   S702_TL_DC_U262_1.Visu_Adv_Arr[14] := FALSE;
   S702_TL_DC_U262_1.Visu_Adv_Arr[15] := FALSE;
   S702_TL_DC_U262_1.Visu_Ret_Arr[0] := FALSE;
   S702_TL_DC_U262_1.Visu_Ret_Arr[1] := FALSE;
   S702_TL_DC_U262_1.Visu_Ret_Arr[2] := FALSE;
   S702_TL_DC_U262_1.Visu_Ret_Arr[3] := FALSE;
   S702_TL_DC_U262_1.Visu_Ret_Arr[4] := FALSE;
   S702_TL_DC_U262_1.Visu_Ret_Arr[5] := FALSE;
   S702_TL_DC_U262_1.Visu_Ret_Arr[6] := FALSE;
   S702_TL_DC_U262_1.Visu_Ret_Arr[7] := FALSE;
   S702_TL_DC_U262_1.Visu_Ret_Arr[8] := FALSE;
   S702_TL_DC_U262_1.Visu_Ret_Arr[9] := FALSE;
   S702_TL_DC_U262_1.Visu_Ret_Arr[10] := FALSE;
   S702_TL_DC_U262_1.Visu_Ret_Arr[11] := FALSE;
   S702_TL_DC_U262_1.Visu_Ret_Arr[12] := FALSE;
   S702_TL_DC_U262_1.Visu_Ret_Arr[13] := FALSE;
   S702_TL_DC_U262_1.Visu_Ret_Arr[14] := FALSE;
   S702_TL_DC_U262_1.Visu_Ret_Arr[15] := FALSE;
   S702_TL_DC_U262_1.BLK_Move_Ret := 0;
   S702_TL_DC_U262_1.Enable := FALSE;
   S702_TL_DC_U262_1.Adv_End := FALSE;
   S702_TL_DC_U262_1.Ret_End := FALSE;
   S702_TL_DC_U262_1_CLAMP.Enable_Aux := FALSE;
   S702_TL_DC_U262_1_CLAMP.Adv_Amount := 0;
   S702_TL_DC_U262_1_CLAMP.Ret_Amount := 0;
   S702_TL_DC_U262_1_CLAMP.LS_Adv1 := FALSE;
   S702_TL_DC_U262_1_CLAMP.LS_Ret1 := FALSE;
   S702_TL_DC_U262_1_CLAMP.LS_Adv2 := FALSE;
   S702_TL_DC_U262_1_CLAMP.LS_Ret2 := FALSE;
   S702_TL_DC_U262_1_CLAMP.LS_Adv3 := FALSE;
   S702_TL_DC_U262_1_CLAMP.LS_Ret3 := FALSE;
   S702_TL_DC_U262_1_CLAMP.LS_Adv4 := FALSE;
   S702_TL_DC_U262_1_CLAMP.LS_Ret4 := FALSE;
   S702_TL_DC_U262_1_CLAMP.LS_Adv5 := FALSE;
   S702_TL_DC_U262_1_CLAMP.LS_Ret5 := FALSE;
   S702_TL_DC_U262_1_CLAMP.LS_Adv6 := FALSE;
   S702_TL_DC_U262_1_CLAMP.LS_Ret6 := FALSE;
   S702_TL_DC_U262_1_CLAMP.LS_Adv7 := FALSE;
   S702_TL_DC_U262_1_CLAMP.LS_Ret7 := FALSE;
   S702_TL_DC_U262_1_CLAMP.LS_Adv8 := FALSE;
   S702_TL_DC_U262_1_CLAMP.LS_Ret8 := FALSE;
   S702_TL_DC_U262_1_CLAMP.SOL_Adv := FALSE;
   S702_TL_DC_U262_1_CLAMP.SOL_Ret := FALSE;
   S702_TL_DC_U262_1_CLAMP.M_Ready := FALSE;
   S702_TL_DC_U262_1_CLAMP.T_CHK1 := T#0MS;
   S702_TL_DC_U262_1_CLAMP.T_CHK2 := T#0MS;
   S702_TL_DC_U262_1_CLAMP.PB_Lamp_CHK := FALSE;
   S702_TL_DC_U262_1_CLAMP.PB_Error_Rst := FALSE;
   S702_TL_DC_U262_1_CLAMP.M_FLICK := FALSE;
   S702_TL_DC_U262_1_CLAMP.M_Adv_Err := FALSE;
   S702_TL_DC_U262_1_CLAMP.M_Ret_Err := FALSE;
   S702_TL_DC_U262_1_CLAMP.LP_Adv := FALSE;
   S702_TL_DC_U262_1_CLAMP.LP_Ret := FALSE;
   S702_TL_DC_U262_1_CLAMP.Visu_Adv := W#16#0;
   S702_TL_DC_U262_1_CLAMP.Visu_Ret := W#16#0;
   S702_TL_DC_U262_1_CLAMP.Error_T1.IN := FALSE;
   S702_TL_DC_U262_1_CLAMP.Error_T1.PT := T#0MS;
   S702_TL_DC_U262_1_CLAMP.Error_T1.Q := FALSE;
   S702_TL_DC_U262_1_CLAMP.Error_T1.ET := T#0MS;
   S702_TL_DC_U262_1_CLAMP.Error_T1.STATE := B#16#0;
   S702_TL_DC_U262_1_CLAMP.Error_T1.STIME := T#0MS;
   S702_TL_DC_U262_1_CLAMP.Error_T1.ATIME := T#0MS;
   S702_TL_DC_U262_1_CLAMP.Error_T2.IN := FALSE;
   S702_TL_DC_U262_1_CLAMP.Error_T2.PT := T#0MS;
   S702_TL_DC_U262_1_CLAMP.Error_T2.Q := FALSE;
   S702_TL_DC_U262_1_CLAMP.Error_T2.ET := T#0MS;
   S702_TL_DC_U262_1_CLAMP.Error_T2.STATE := B#16#0;
   S702_TL_DC_U262_1_CLAMP.Error_T2.STIME := T#0MS;
   S702_TL_DC_U262_1_CLAMP.Error_T2.ATIME := T#0MS;
   S702_TL_DC_U262_1_CLAMP.Adv_End_Aux := FALSE;
   S702_TL_DC_U262_1_CLAMP.Ret_End_Aux := FALSE;
   S702_TL_DC_U262_1_CLAMP.CHK_Aux1 := FALSE;
   S702_TL_DC_U262_1_CLAMP.CHK_Aux2 := FALSE;
   S702_TL_DC_U262_1_CLAMP.Error_T1_DN := FALSE;
   S702_TL_DC_U262_1_CLAMP.Error_T2_DN := FALSE;
   S702_TL_DC_U262_1_CLAMP.Adv_Memo := FALSE;
   S702_TL_DC_U262_1_CLAMP.Visu_Adv_Arr[0] := FALSE;
   S702_TL_DC_U262_1_CLAMP.Visu_Adv_Arr[1] := FALSE;
   S702_TL_DC_U262_1_CLAMP.Visu_Adv_Arr[2] := FALSE;
   S702_TL_DC_U262_1_CLAMP.Visu_Adv_Arr[3] := FALSE;
   S702_TL_DC_U262_1_CLAMP.Visu_Adv_Arr[4] := FALSE;
   S702_TL_DC_U262_1_CLAMP.Visu_Adv_Arr[5] := FALSE;
   S702_TL_DC_U262_1_CLAMP.Visu_Adv_Arr[6] := FALSE;
   S702_TL_DC_U262_1_CLAMP.Visu_Adv_Arr[7] := FALSE;
   S702_TL_DC_U262_1_CLAMP.Visu_Adv_Arr[8] := FALSE;
   S702_TL_DC_U262_1_CLAMP.Visu_Adv_Arr[9] := FALSE;
   S702_TL_DC_U262_1_CLAMP.Visu_Adv_Arr[10] := FALSE;
   S702_TL_DC_U262_1_CLAMP.Visu_Adv_Arr[11] := FALSE;
   S702_TL_DC_U262_1_CLAMP.Visu_Adv_Arr[12] := FALSE;
   S702_TL_DC_U262_1_CLAMP.Visu_Adv_Arr[13] := FALSE;
   S702_TL_DC_U262_1_CLAMP.Visu_Adv_Arr[14] := FALSE;
   S702_TL_DC_U262_1_CLAMP.Visu_Adv_Arr[15] := FALSE;
   S702_TL_DC_U262_1_CLAMP.Visu_Ret_Arr[0] := FALSE;
   S702_TL_DC_U262_1_CLAMP.Visu_Ret_Arr[1] := FALSE;
   S702_TL_DC_U262_1_CLAMP.Visu_Ret_Arr[2] := FALSE;
   S702_TL_DC_U262_1_CLAMP.Visu_Ret_Arr[3] := FALSE;
   S702_TL_DC_U262_1_CLAMP.Visu_Ret_Arr[4] := FALSE;
   S702_TL_DC_U262_1_CLAMP.Visu_Ret_Arr[5] := FALSE;
   S702_TL_DC_U262_1_CLAMP.Visu_Ret_Arr[6] := FALSE;
   S702_TL_DC_U262_1_CLAMP.Visu_Ret_Arr[7] := FALSE;
   S702_TL_DC_U262_1_CLAMP.Visu_Ret_Arr[8] := FALSE;
   S702_TL_DC_U262_1_CLAMP.Visu_Ret_Arr[9] := FALSE;
   S702_TL_DC_U262_1_CLAMP.Visu_Ret_Arr[10] := FALSE;
   S702_TL_DC_U262_1_CLAMP.Visu_Ret_Arr[11] := FALSE;
   S702_TL_DC_U262_1_CLAMP.Visu_Ret_Arr[12] := FALSE;
   S702_TL_DC_U262_1_CLAMP.Visu_Ret_Arr[13] := FALSE;
   S702_TL_DC_U262_1_CLAMP.Visu_Ret_Arr[14] := FALSE;
   S702_TL_DC_U262_1_CLAMP.Visu_Ret_Arr[15] := FALSE;
   S702_TL_DC_U262_1_CLAMP.BLK_Move_Ret := 0;
   S702_TL_DC_U262_1_CLAMP.Enable := FALSE;
   S702_TL_DC_U262_1_CLAMP.Adv_End := FALSE;
   S702_TL_DC_U262_1_CLAMP.Ret_End := FALSE;
   S702_TL_DC_U261_2_CLAMP.Enable_Aux := FALSE;
   S702_TL_DC_U261_2_CLAMP.Adv_Amount := 0;
   S702_TL_DC_U261_2_CLAMP.Ret_Amount := 0;
   S702_TL_DC_U261_2_CLAMP.LS_Adv1 := FALSE;
   S702_TL_DC_U261_2_CLAMP.LS_Ret1 := FALSE;
   S702_TL_DC_U261_2_CLAMP.LS_Adv2 := FALSE;
   S702_TL_DC_U261_2_CLAMP.LS_Ret2 := FALSE;
   S702_TL_DC_U261_2_CLAMP.LS_Adv3 := FALSE;
   S702_TL_DC_U261_2_CLAMP.LS_Ret3 := FALSE;
   S702_TL_DC_U261_2_CLAMP.LS_Adv4 := FALSE;
   S702_TL_DC_U261_2_CLAMP.LS_Ret4 := FALSE;
   S702_TL_DC_U261_2_CLAMP.LS_Adv5 := FALSE;
   S702_TL_DC_U261_2_CLAMP.LS_Ret5 := FALSE;
   S702_TL_DC_U261_2_CLAMP.LS_Adv6 := FALSE;
   S702_TL_DC_U261_2_CLAMP.LS_Ret6 := FALSE;
   S702_TL_DC_U261_2_CLAMP.LS_Adv7 := FALSE;
   S702_TL_DC_U261_2_CLAMP.LS_Ret7 := FALSE;
   S702_TL_DC_U261_2_CLAMP.LS_Adv8 := FALSE;
   S702_TL_DC_U261_2_CLAMP.LS_Ret8 := FALSE;
   S702_TL_DC_U261_2_CLAMP.SOL_Adv := FALSE;
   S702_TL_DC_U261_2_CLAMP.SOL_Ret := FALSE;
   S702_TL_DC_U261_2_CLAMP.M_Ready := FALSE;
   S702_TL_DC_U261_2_CLAMP.T_CHK1 := T#0MS;
   S702_TL_DC_U261_2_CLAMP.T_CHK2 := T#0MS;
   S702_TL_DC_U261_2_CLAMP.PB_Lamp_CHK := FALSE;
   S702_TL_DC_U261_2_CLAMP.PB_Error_Rst := FALSE;
   S702_TL_DC_U261_2_CLAMP.M_FLICK := FALSE;
   S702_TL_DC_U261_2_CLAMP.M_Adv_Err := FALSE;
   S702_TL_DC_U261_2_CLAMP.M_Ret_Err := FALSE;
   S702_TL_DC_U261_2_CLAMP.LP_Adv := FALSE;
   S702_TL_DC_U261_2_CLAMP.LP_Ret := FALSE;
   S702_TL_DC_U261_2_CLAMP.Visu_Adv := W#16#0;
   S702_TL_DC_U261_2_CLAMP.Visu_Ret := W#16#0;
   S702_TL_DC_U261_2_CLAMP.Error_T1.IN := FALSE;
   S702_TL_DC_U261_2_CLAMP.Error_T1.PT := T#0MS;
   S702_TL_DC_U261_2_CLAMP.Error_T1.Q := FALSE;
   S702_TL_DC_U261_2_CLAMP.Error_T1.ET := T#0MS;
   S702_TL_DC_U261_2_CLAMP.Error_T1.STATE := B#16#0;
   S702_TL_DC_U261_2_CLAMP.Error_T1.STIME := T#0MS;
   S702_TL_DC_U261_2_CLAMP.Error_T1.ATIME := T#0MS;
   S702_TL_DC_U261_2_CLAMP.Error_T2.IN := FALSE;
   S702_TL_DC_U261_2_CLAMP.Error_T2.PT := T#0MS;
   S702_TL_DC_U261_2_CLAMP.Error_T2.Q := FALSE;
   S702_TL_DC_U261_2_CLAMP.Error_T2.ET := T#0MS;
   S702_TL_DC_U261_2_CLAMP.Error_T2.STATE := B#16#0;
   S702_TL_DC_U261_2_CLAMP.Error_T2.STIME := T#0MS;
   S702_TL_DC_U261_2_CLAMP.Error_T2.ATIME := T#0MS;
   S702_TL_DC_U261_2_CLAMP.Adv_End_Aux := FALSE;
   S702_TL_DC_U261_2_CLAMP.Ret_End_Aux := FALSE;
   S702_TL_DC_U261_2_CLAMP.CHK_Aux1 := FALSE;
   S702_TL_DC_U261_2_CLAMP.CHK_Aux2 := FALSE;
   S702_TL_DC_U261_2_CLAMP.Error_T1_DN := FALSE;
   S702_TL_DC_U261_2_CLAMP.Error_T2_DN := FALSE;
   S702_TL_DC_U261_2_CLAMP.Adv_Memo := FALSE;
   S702_TL_DC_U261_2_CLAMP.Visu_Adv_Arr[0] := FALSE;
   S702_TL_DC_U261_2_CLAMP.Visu_Adv_Arr[1] := FALSE;
   S702_TL_DC_U261_2_CLAMP.Visu_Adv_Arr[2] := FALSE;
   S702_TL_DC_U261_2_CLAMP.Visu_Adv_Arr[3] := FALSE;
   S702_TL_DC_U261_2_CLAMP.Visu_Adv_Arr[4] := FALSE;
   S702_TL_DC_U261_2_CLAMP.Visu_Adv_Arr[5] := FALSE;
   S702_TL_DC_U261_2_CLAMP.Visu_Adv_Arr[6] := FALSE;
   S702_TL_DC_U261_2_CLAMP.Visu_Adv_Arr[7] := FALSE;
   S702_TL_DC_U261_2_CLAMP.Visu_Adv_Arr[8] := FALSE;
   S702_TL_DC_U261_2_CLAMP.Visu_Adv_Arr[9] := FALSE;
   S702_TL_DC_U261_2_CLAMP.Visu_Adv_Arr[10] := FALSE;
   S702_TL_DC_U261_2_CLAMP.Visu_Adv_Arr[11] := FALSE;
   S702_TL_DC_U261_2_CLAMP.Visu_Adv_Arr[12] := FALSE;
   S702_TL_DC_U261_2_CLAMP.Visu_Adv_Arr[13] := FALSE;
   S702_TL_DC_U261_2_CLAMP.Visu_Adv_Arr[14] := FALSE;
   S702_TL_DC_U261_2_CLAMP.Visu_Adv_Arr[15] := FALSE;
   S702_TL_DC_U261_2_CLAMP.Visu_Ret_Arr[0] := FALSE;
   S702_TL_DC_U261_2_CLAMP.Visu_Ret_Arr[1] := FALSE;
   S702_TL_DC_U261_2_CLAMP.Visu_Ret_Arr[2] := FALSE;
   S702_TL_DC_U261_2_CLAMP.Visu_Ret_Arr[3] := FALSE;
   S702_TL_DC_U261_2_CLAMP.Visu_Ret_Arr[4] := FALSE;
   S702_TL_DC_U261_2_CLAMP.Visu_Ret_Arr[5] := FALSE;
   S702_TL_DC_U261_2_CLAMP.Visu_Ret_Arr[6] := FALSE;
   S702_TL_DC_U261_2_CLAMP.Visu_Ret_Arr[7] := FALSE;
   S702_TL_DC_U261_2_CLAMP.Visu_Ret_Arr[8] := FALSE;
   S702_TL_DC_U261_2_CLAMP.Visu_Ret_Arr[9] := FALSE;
   S702_TL_DC_U261_2_CLAMP.Visu_Ret_Arr[10] := FALSE;
   S702_TL_DC_U261_2_CLAMP.Visu_Ret_Arr[11] := FALSE;
   S702_TL_DC_U261_2_CLAMP.Visu_Ret_Arr[12] := FALSE;
   S702_TL_DC_U261_2_CLAMP.Visu_Ret_Arr[13] := FALSE;
   S702_TL_DC_U261_2_CLAMP.Visu_Ret_Arr[14] := FALSE;
   S702_TL_DC_U261_2_CLAMP.Visu_Ret_Arr[15] := FALSE;
   S702_TL_DC_U261_2_CLAMP.BLK_Move_Ret := 0;
   S702_TL_DC_U261_2_CLAMP.Enable := FALSE;
   S702_TL_DC_U261_2_CLAMP.Adv_End := FALSE;
   S702_TL_DC_U261_2_CLAMP.Ret_End := FALSE;
END_DATA_BLOCK

FUNCTION FC 124 : VOID
TITLE =
VERSION : 0.1

BEGIN
NETWORK
TITLE =
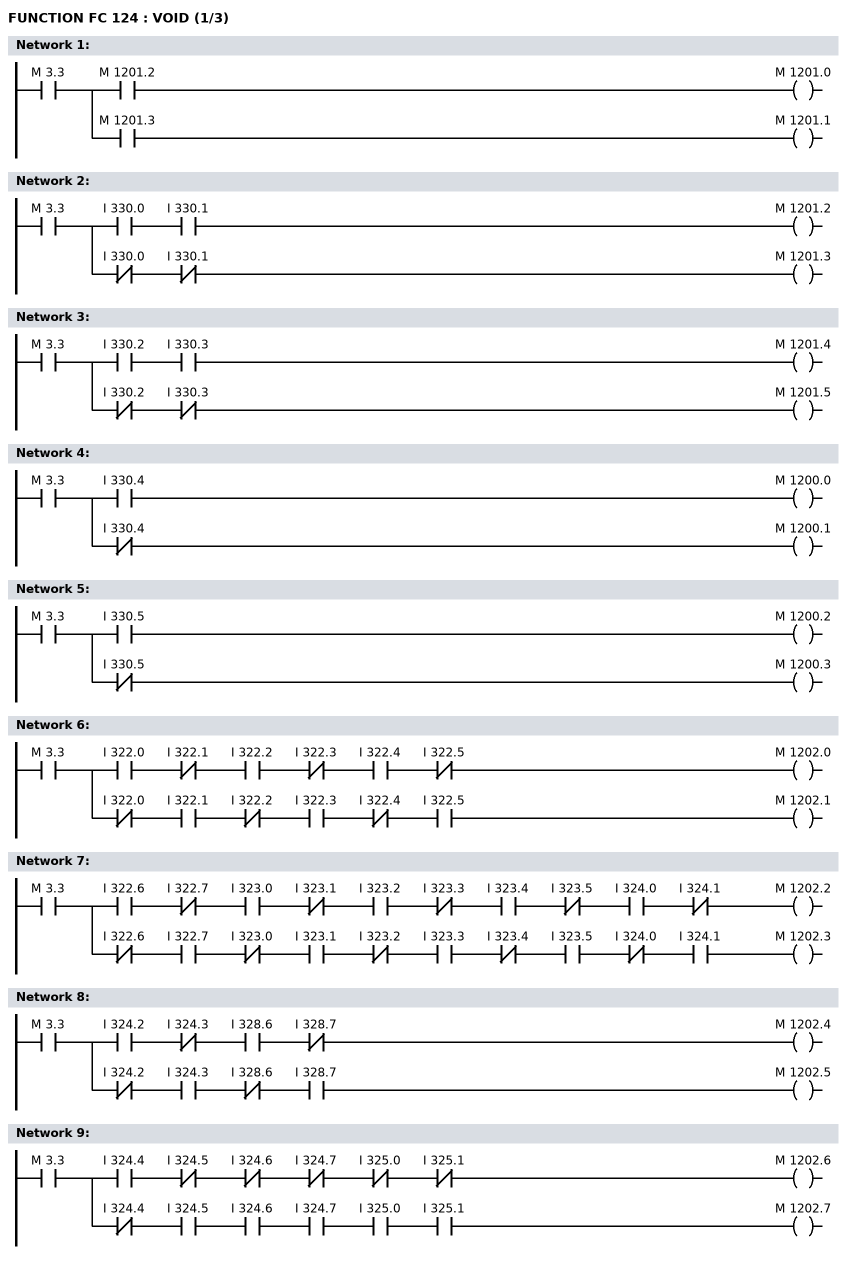

      A     M      3.3;
      =     L      0.0;
      A     L      0.0;
      A     M   1201.2;
      =     M   1201.0;
      A     L      0.0;
      A     M   1201.3;
      =     M   1201.1;
NETWORK
TITLE =

      A     M      3.3;
      =     L      0.0;
      A     L      0.0;
      A     I    330.0;
      A     I    330.1;
      =     M   1201.2;
      A     L      0.0;
      AN    I    330.0;
      AN    I    330.1;
      =     M   1201.3;
NETWORK
TITLE =

      A     M      3.3;
      =     L      0.0;
      A     L      0.0;
      A     I    330.2;
      A     I    330.3;
      =     M   1201.4;
      A     L      0.0;
      AN    I    330.2;
      AN    I    330.3;
      =     M   1201.5;
NETWORK
TITLE =

      A     M      3.3;
      =     L      0.0;
      A     L      0.0;
      A     I    330.4;
      =     M   1200.0;
      A     L      0.0;
      AN    I    330.4;
      =     M   1200.1;
NETWORK
TITLE =

      A     M      3.3;
      =     L      0.0;
      A     L      0.0;
      A     I    330.5;
      =     M   1200.2;
      A     L      0.0;
      AN    I    330.5;
      =     M   1200.3;
NETWORK
TITLE =

      A     M      3.3;
      =     L      0.0;
      A     L      0.0;
      A     I    322.0;
      AN    I    322.1;
      A     I    322.2;
      AN    I    322.3;
      A     I    322.4;
      AN    I    322.5;
      =     M   1202.0;
      A     L      0.0;
      AN    I    322.0;
      A     I    322.1;
      AN    I    322.2;
      A     I    322.3;
      AN    I    322.4;
      A     I    322.5;
      =     M   1202.1;
NETWORK
TITLE =

      A     M      3.3;
      =     L      0.0;
      A     L      0.0;
      A     I    322.6;
      AN    I    322.7;
      A     I    323.0;
      AN    I    323.1;
      A     I    323.2;
      AN    I    323.3;
      A     I    323.4;
      AN    I    323.5;
      A     I    324.0;
      AN    I    324.1;
      =     M   1202.2;
      A     L      0.0;
      AN    I    322.6;
      A     I    322.7;
      AN    I    323.0;
      A     I    323.1;
      AN    I    323.2;
      A     I    323.3;
      AN    I    323.4;
      A     I    323.5;
      AN    I    324.0;
      A     I    324.1;
      =     M   1202.3;
NETWORK
TITLE =

      A     M      3.3;
      =     L      0.0;
      A     L      0.0;
      A     I    324.2;
      AN    I    324.3;
      A     I    328.6;
      AN    I    328.7;
      =     M   1202.4;
      A     L      0.0;
      AN    I    324.2;
      A     I    324.3;
      AN    I    328.6;
      A     I    328.7;
      =     M   1202.5;
NETWORK
TITLE =

      A     M      3.3;
      =     L      0.0;
      A     L      0.0;
      A     I    324.4;
      AN    I    324.5;
      AN    I    324.6;
      AN    I    324.7;
      AN    I    325.0;
      AN    I    325.1;
      =     M   1202.6;
      A     L      0.0;
      AN    I    324.4;
      A     I    324.5;
      A     I    324.6;
      A     I    324.7;
      A     I    325.0;
      A     I    325.1;
      =     M   1202.7;
NETWORK
TITLE =
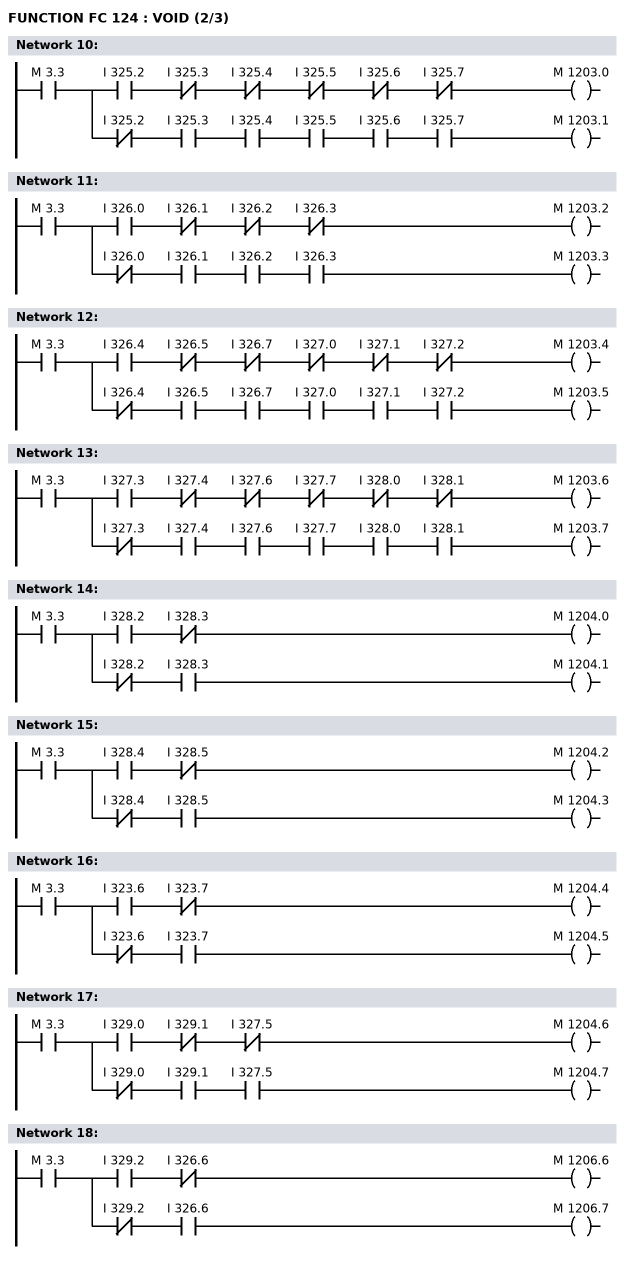

      A     M      3.3;
      =     L      0.0;
      A     L      0.0;
      A     I    325.2;
      AN    I    325.3;
      AN    I    325.4;
      AN    I    325.5;
      AN    I    325.6;
      AN    I    325.7;
      =     M   1203.0;
      A     L      0.0;
      AN    I    325.2;
      A     I    325.3;
      A     I    325.4;
      A     I    325.5;
      A     I    325.6;
      A     I    325.7;
      =     M   1203.1;
NETWORK
TITLE =

      A     M      3.3;
      =     L      0.0;
      A     L      0.0;
      A     I    326.0;
      AN    I    326.1;
      AN    I    326.2;
      AN    I    326.3;
      =     M   1203.2;
      A     L      0.0;
      AN    I    326.0;
      A     I    326.1;
      A     I    326.2;
      A     I    326.3;
      =     M   1203.3;
NETWORK
TITLE =

      A     M      3.3;
      =     L      0.0;
      A     L      0.0;
      A     I    326.4;
      AN    I    326.5;
      AN    I    326.7;
      AN    I    327.0;
      AN    I    327.1;
      AN    I    327.2;
      =     M   1203.4;
      A     L      0.0;
      AN    I    326.4;
      A     I    326.5;
      A     I    326.7;
      A     I    327.0;
      A     I    327.1;
      A     I    327.2;
      =     M   1203.5;
NETWORK
TITLE =

      A     M      3.3;
      =     L      0.0;
      A     L      0.0;
      A     I    327.3;
      AN    I    327.4;
      AN    I    327.6;
      AN    I    327.7;
      AN    I    328.0;
      AN    I    328.1;
      =     M   1203.6;
      A     L      0.0;
      AN    I    327.3;
      A     I    327.4;
      A     I    327.6;
      A     I    327.7;
      A     I    328.0;
      A     I    328.1;
      =     M   1203.7;
NETWORK
TITLE =

      A     M      3.3;
      =     L      0.0;
      A     L      0.0;
      A     I    328.2;
      AN    I    328.3;
      =     M   1204.0;
      A     L      0.0;
      AN    I    328.2;
      A     I    328.3;
      =     M   1204.1;
NETWORK
TITLE =

      A     M      3.3;
      =     L      0.0;
      A     L      0.0;
      A     I    328.4;
      AN    I    328.5;
      =     M   1204.2;
      A     L      0.0;
      AN    I    328.4;
      A     I    328.5;
      =     M   1204.3;
NETWORK
TITLE =

      A     M      3.3;
      =     L      0.0;
      A     L      0.0;
      A     I    323.6;
      AN    I    323.7;
      =     M   1204.4;
      A     L      0.0;
      AN    I    323.6;
      A     I    323.7;
      =     M   1204.5;
NETWORK
TITLE =

      A     M      3.3;
      =     L      0.0;
      A     L      0.0;
      A     I    329.0;
      AN    I    329.1;
      AN    I    327.5;
      =     M   1204.6;
      A     L      0.0;
      AN    I    329.0;
      A     I    329.1;
      A     I    327.5;
      =     M   1204.7;
NETWORK
TITLE =

      A     M      3.3;
      =     L      0.0;
      A     L      0.0;
      A     I    329.2;
      AN    I    326.6;
      =     M   1206.6;
      A     L      0.0;
      AN    I    329.2;
      A     I    326.6;
      =     M   1206.7;
NETWORK
TITLE =
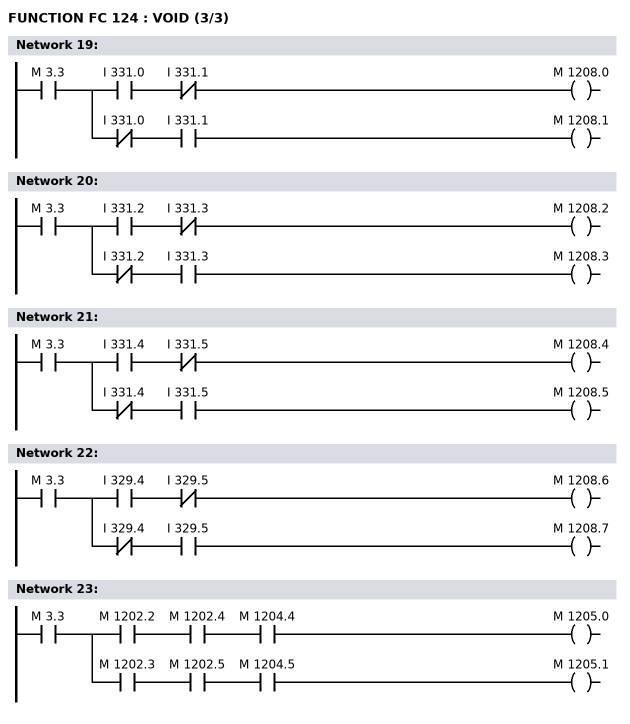

      A     M      3.3;
      =     L      0.0;
      A     L      0.0;
      A     I    331.0;
      AN    I    331.1;
      =     M   1208.0;
      A     L      0.0;
      AN    I    331.0;
      A     I    331.1;
      =     M   1208.1;
NETWORK
TITLE =

      A     M      3.3;
      =     L      0.0;
      A     L      0.0;
      A     I    331.2;
      AN    I    331.3;
      =     M   1208.2;
      A     L      0.0;
      AN    I    331.2;
      A     I    331.3;
      =     M   1208.3;
NETWORK
TITLE =

      A     M      3.3;
      =     L      0.0;
      A     L      0.0;
      A     I    331.4;
      AN    I    331.5;
      =     M   1208.4;
      A     L      0.0;
      AN    I    331.4;
      A     I    331.5;
      =     M   1208.5;
NETWORK
TITLE =

      A     M      3.3;
      =     L      0.0;
      A     L      0.0;
      A     I    329.4;
      AN    I    329.5;
      =     M   1208.6;
      A     L      0.0;
      AN    I    329.4;
      A     I    329.5;
      =     M   1208.7;
NETWORK
TITLE =

      A     M      3.3;
      =     L      0.0;
      A     L      0.0;
      A     M   1202.2;
      A     M   1202.4;
      A     M   1204.4;
      =     M   1205.0;
      A     L      0.0;
      A     M   1202.3;
      A     M   1202.5;
      A     M   1204.5;
      =     M   1205.1;
NETWORK
TITLE =

      A     M      3.3;
      =     L      0.0;
      A     L      0.0;
      A     M   1202.6;
      A     M   1203.0;
      A     M   1203.2;
      A     M   1203.4;
      A     M   1203.6;
      A     M   1206.6;
      =     L      0.1;
      A     L      0.1;
      BLD   102;
      =     M   1205.2;
      A     L      0.1;
      A     M   1204.2;
      A     M   1204.6;
      =     M   1205.4;
      A     L      0.0;
      A     M   1202.7;
      A     M   1203.1;
      A     M   1203.3;
      A     M   1203.5;
      A     M   1203.7;
      A     M   1206.7;
      =     L      0.1;
      A     L      0.1;
      BLD   102;
      =     M   1205.3;
      A     L      0.1;
      A     M   1204.3;
      A     M   1204.7;
      =     M   1205.5;
NETWORK
TITLE =
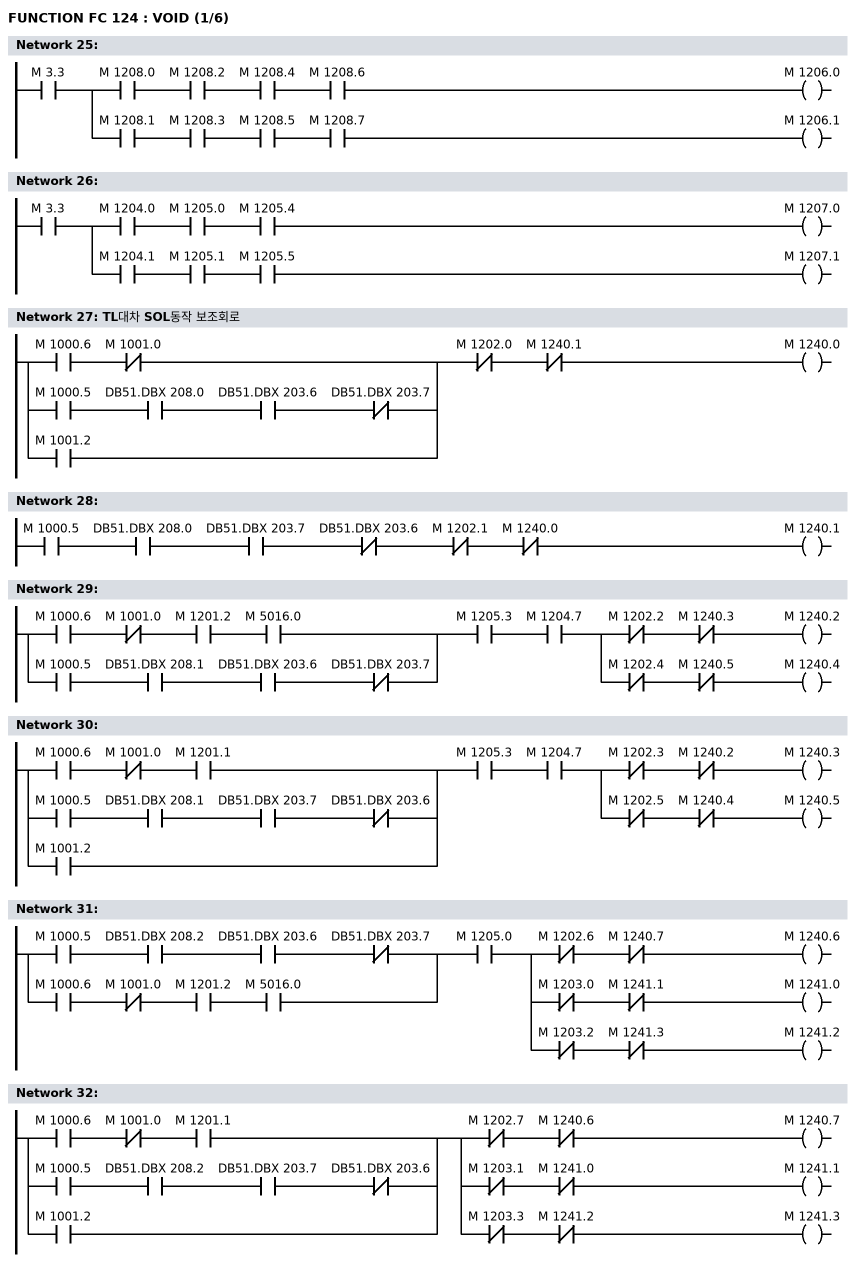

      A     M      3.3;
      =     L      0.0;
      A     L      0.0;
      A     M   1208.0;
      A     M   1208.2;
      A     M   1208.4;
      A     M   1208.6;
      =     M   1206.0;
      A     L      0.0;
      A     M   1208.1;
      A     M   1208.3;
      A     M   1208.5;
      A     M   1208.7;
      =     M   1206.1;
NETWORK
TITLE =

      A     M      3.3;
      =     L      0.0;
      A     L      0.0;
      A     M   1204.0;
      A     M   1205.0;
      A     M   1205.4;
      =     M   1207.0;
      A     L      0.0;
      A     M   1204.1;
      A     M   1205.1;
      A     M   1205.5;
      =     M   1207.1;
NETWORK
TITLE =TL대차 SOL동작 보조회로

      A(    ;
      A     M   1000.6;
      AN    M   1001.0;
      O     ;
      A     M   1000.5;
      A     DB51.DBX  208.0;
      A     DB51.DBX  203.6;
      AN    DB51.DBX  203.7;
      O     M   1001.2;
      )     ;
      AN    M   1202.0;
      AN    M   1240.1;
      =     M   1240.0;
NETWORK
TITLE =

      A     M   1000.5;
      A     DB51.DBX  208.0;
      A     DB51.DBX  203.7;
      AN    DB51.DBX  203.6;
      AN    M   1202.1;
      AN    M   1240.0;
      =     M   1240.1;
NETWORK
TITLE =

      A(    ;
      A     M   1000.6;
      AN    M   1001.0;
      A     M   1201.2;
      A     M   5016.0;
      O     ;
      A     M   1000.5;
      A     DB51.DBX  208.1;
      A     DB51.DBX  203.6;
      AN    DB51.DBX  203.7;
      )     ;
      A     M   1205.3;
      A     M   1204.7;
      =     L      0.0;
      A     L      0.0;
      AN    M   1202.2;
      AN    M   1240.3;
      =     M   1240.2;
      A     L      0.0;
      AN    M   1202.4;
      AN    M   1240.5;
      =     M   1240.4;
NETWORK
TITLE =

      A(    ;
      A     M   1000.6;
      AN    M   1001.0;
      A     M   1201.1;
      O     ;
      A     M   1000.5;
      A     DB51.DBX  208.1;
      A     DB51.DBX  203.7;
      AN    DB51.DBX  203.6;
      O     M   1001.2;
      )     ;
      A     M   1205.3;
      A     M   1204.7;
      =     L      0.0;
      A     L      0.0;
      AN    M   1202.3;
      AN    M   1240.2;
      =     M   1240.3;
      A     L      0.0;
      AN    M   1202.5;
      AN    M   1240.4;
      =     M   1240.5;
NETWORK
TITLE =

      A(    ;
      A     M   1000.5;
      A     DB51.DBX  208.2;
      A     DB51.DBX  203.6;
      AN    DB51.DBX  203.7;
      O     ;
      A     M   1000.6;
      AN    M   1001.0;
      A     M   1201.2;
      A     M   5016.0;
      )     ;
      A     M   1205.0;
      =     L      0.0;
      A     L      0.0;
      AN    M   1202.6;
      AN    M   1240.7;
      =     M   1240.6;
      A     L      0.0;
      AN    M   1203.0;
      AN    M   1241.1;
      =     M   1241.0;
      A     L      0.0;
      AN    M   1203.2;
      AN    M   1241.3;
      =     M   1241.2;
NETWORK
TITLE =

      A     M   1000.6;
      AN    M   1001.0;
      A     M   1201.1;
      O     ;
      A     M   1000.5;
      A     DB51.DBX  208.2;
      A     DB51.DBX  203.7;
      AN    DB51.DBX  203.6;
      O     M   1001.2;
      =     L      0.0;
      A     L      0.0;
      AN    M   1202.7;
      AN    M   1240.6;
      =     M   1240.7;
      A     L      0.0;
      AN    M   1203.1;
      AN    M   1241.0;
      =     M   1241.1;
      A     L      0.0;
      AN    M   1203.3;
      AN    M   1241.2;
      =     M   1241.3;
NETWORK
TITLE =
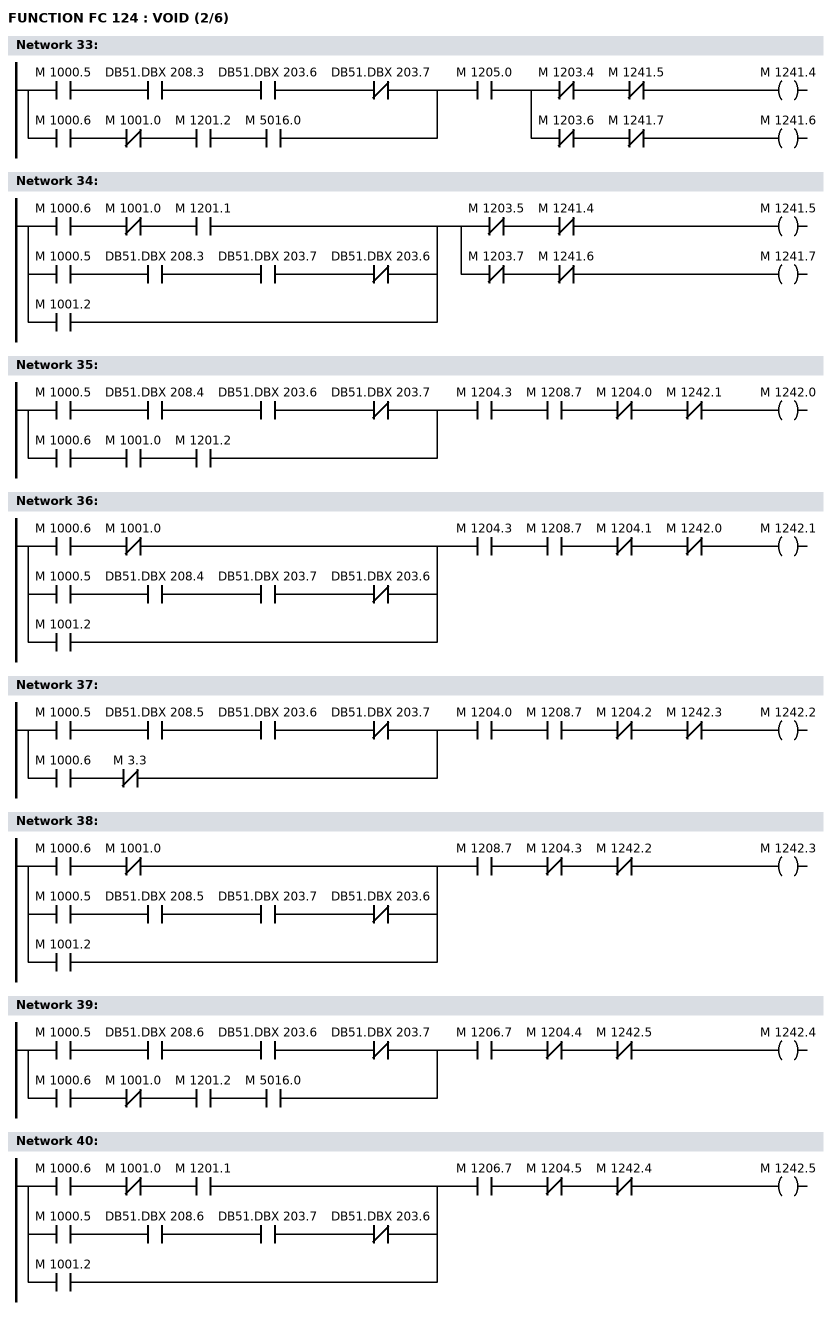

      A(    ;
      A     M   1000.5;
      A     DB51.DBX  208.3;
      A     DB51.DBX  203.6;
      AN    DB51.DBX  203.7;
      O     ;
      A     M   1000.6;
      AN    M   1001.0;
      A     M   1201.2;
      A     M   5016.0;
      )     ;
      A     M   1205.0;
      =     L      0.0;
      A     L      0.0;
      AN    M   1203.4;
      AN    M   1241.5;
      =     M   1241.4;
      A     L      0.0;
      AN    M   1203.6;
      AN    M   1241.7;
      =     M   1241.6;
NETWORK
TITLE =

      A     M   1000.6;
      AN    M   1001.0;
      A     M   1201.1;
      O     ;
      A     M   1000.5;
      A     DB51.DBX  208.3;
      A     DB51.DBX  203.7;
      AN    DB51.DBX  203.6;
      O     M   1001.2;
      =     L      0.0;
      A     L      0.0;
      AN    M   1203.5;
      AN    M   1241.4;
      =     M   1241.5;
      A     L      0.0;
      AN    M   1203.7;
      AN    M   1241.6;
      =     M   1241.7;
NETWORK
TITLE =

      A(    ;
      A     M   1000.5;
      A     DB51.DBX  208.4;
      A     DB51.DBX  203.6;
      AN    DB51.DBX  203.7;
      O     ;
      A     M   1000.6;
      A     M   1001.0;
      A     M   1201.2;
      )     ;
      A     M   1204.3;
      A     M   1208.7;
      AN    M   1204.0;
      AN    M   1242.1;
      =     M   1242.0;
NETWORK
TITLE =

      A(    ;
      A     M   1000.6;
      AN    M   1001.0;
      O     ;
      A     M   1000.5;
      A     DB51.DBX  208.4;
      A     DB51.DBX  203.7;
      AN    DB51.DBX  203.6;
      O     M   1001.2;
      )     ;
      A     M   1204.3;
      A     M   1208.7;
      AN    M   1204.1;
      AN    M   1242.0;
      =     M   1242.1;
NETWORK
TITLE =

      A(    ;
      A     M   1000.5;
      A     DB51.DBX  208.5;
      A     DB51.DBX  203.6;
      AN    DB51.DBX  203.7;
      O     ;
      A     M   1000.6;
      AN    M      3.3;
      )     ;
      A     M   1204.0;
      A     M   1208.7;
      AN    M   1204.2;
      AN    M   1242.3;
      =     M   1242.2;
NETWORK
TITLE =

      A(    ;
      A     M   1000.6;
      AN    M   1001.0;
      O     ;
      A     M   1000.5;
      A     DB51.DBX  208.5;
      A     DB51.DBX  203.7;
      AN    DB51.DBX  203.6;
      O     M   1001.2;
      )     ;
      A     M   1208.7;
      AN    M   1204.3;
      AN    M   1242.2;
      =     M   1242.3;
NETWORK
TITLE =

      A(    ;
      A     M   1000.5;
      A     DB51.DBX  208.6;
      A     DB51.DBX  203.6;
      AN    DB51.DBX  203.7;
      O     ;
      A     M   1000.6;
      AN    M   1001.0;
      A     M   1201.2;
      A     M   5016.0;
      )     ;
      A     M   1206.7;
      AN    M   1204.4;
      AN    M   1242.5;
      =     M   1242.4;
NETWORK
TITLE =

      A(    ;
      A     M   1000.6;
      AN    M   1001.0;
      A     M   1201.1;
      O     ;
      A     M   1000.5;
      A     DB51.DBX  208.6;
      A     DB51.DBX  203.7;
      AN    DB51.DBX  203.6;
      O     M   1001.2;
      )     ;
      A     M   1206.7;
      AN    M   1204.5;
      AN    M   1242.4;
      =     M   1242.5;
NETWORK
TITLE =
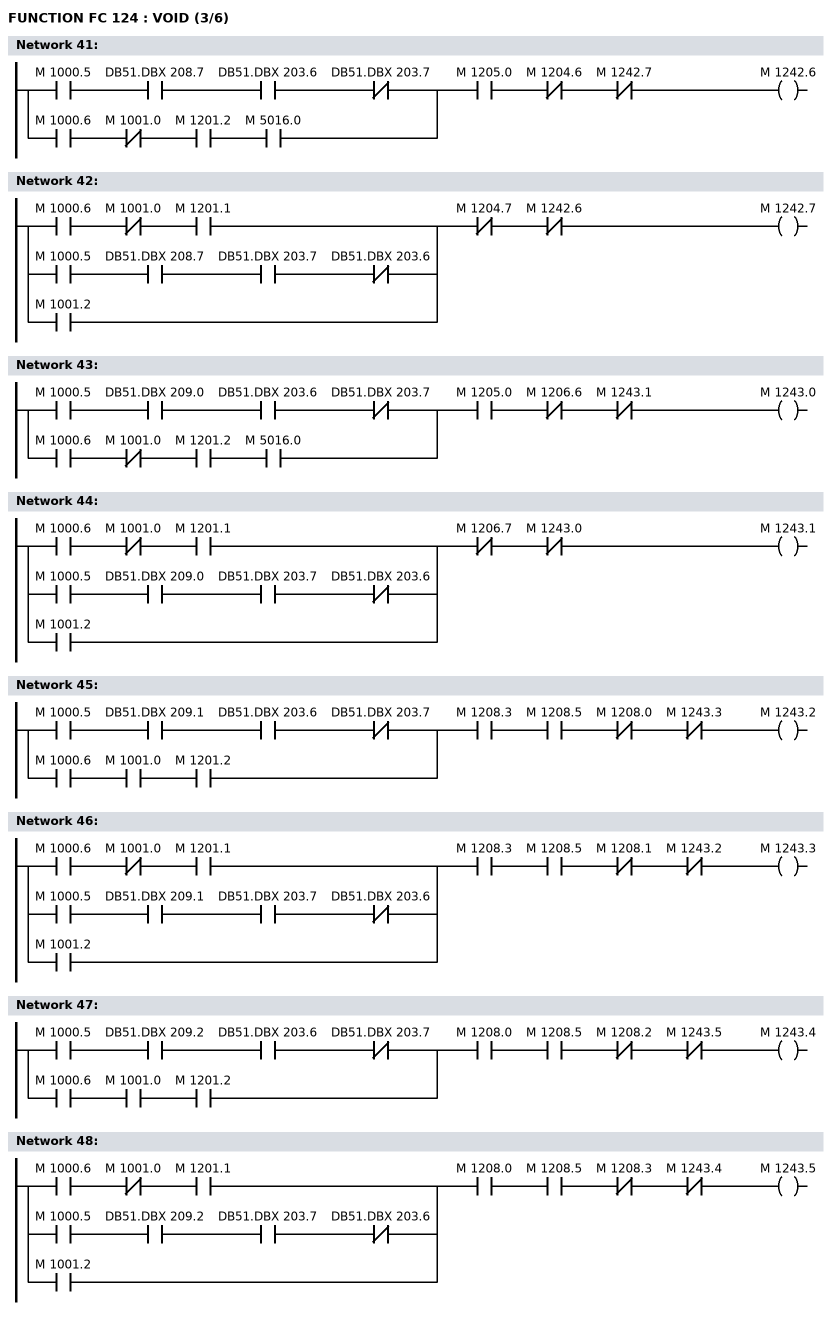

      A(    ;
      A     M   1000.5;
      A     DB51.DBX  208.7;
      A     DB51.DBX  203.6;
      AN    DB51.DBX  203.7;
      O     ;
      A     M   1000.6;
      AN    M   1001.0;
      A     M   1201.2;
      A     M   5016.0;
      )     ;
      A     M   1205.0;
      AN    M   1204.6;
      AN    M   1242.7;
      =     M   1242.6;
NETWORK
TITLE =

      A(    ;
      A     M   1000.6;
      AN    M   1001.0;
      A     M   1201.1;
      O     ;
      A     M   1000.5;
      A     DB51.DBX  208.7;
      A     DB51.DBX  203.7;
      AN    DB51.DBX  203.6;
      O     M   1001.2;
      )     ;
      AN    M   1204.7;
      AN    M   1242.6;
      =     M   1242.7;
NETWORK
TITLE =

      A(    ;
      A     M   1000.5;
      A     DB51.DBX  209.0;
      A     DB51.DBX  203.6;
      AN    DB51.DBX  203.7;
      O     ;
      A     M   1000.6;
      AN    M   1001.0;
      A     M   1201.2;
      A     M   5016.0;
      )     ;
      A     M   1205.0;
      AN    M   1206.6;
      AN    M   1243.1;
      =     M   1243.0;
NETWORK
TITLE =

      A(    ;
      A     M   1000.6;
      AN    M   1001.0;
      A     M   1201.1;
      O     ;
      A     M   1000.5;
      A     DB51.DBX  209.0;
      A     DB51.DBX  203.7;
      AN    DB51.DBX  203.6;
      O     M   1001.2;
      )     ;
      AN    M   1206.7;
      AN    M   1243.0;
      =     M   1243.1;
NETWORK
TITLE =

      A(    ;
      A     M   1000.5;
      A     DB51.DBX  209.1;
      A     DB51.DBX  203.6;
      AN    DB51.DBX  203.7;
      O     ;
      A     M   1000.6;
      A     M   1001.0;
      A     M   1201.2;
      )     ;
      A     M   1208.3;
      A     M   1208.5;
      AN    M   1208.0;
      AN    M   1243.3;
      =     M   1243.2;
NETWORK
TITLE =

      A(    ;
      A     M   1000.6;
      AN    M   1001.0;
      A     M   1201.1;
      O     ;
      A     M   1000.5;
      A     DB51.DBX  209.1;
      A     DB51.DBX  203.7;
      AN    DB51.DBX  203.6;
      O     M   1001.2;
      )     ;
      A     M   1208.3;
      A     M   1208.5;
      AN    M   1208.1;
      AN    M   1243.2;
      =     M   1243.3;
NETWORK
TITLE =

      A(    ;
      A     M   1000.5;
      A     DB51.DBX  209.2;
      A     DB51.DBX  203.6;
      AN    DB51.DBX  203.7;
      O     ;
      A     M   1000.6;
      A     M   1001.0;
      A     M   1201.2;
      )     ;
      A     M   1208.0;
      A     M   1208.5;
      AN    M   1208.2;
      AN    M   1243.5;
      =     M   1243.4;
NETWORK
TITLE =

      A(    ;
      A     M   1000.6;
      AN    M   1001.0;
      A     M   1201.1;
      O     ;
      A     M   1000.5;
      A     DB51.DBX  209.2;
      A     DB51.DBX  203.7;
      AN    DB51.DBX  203.6;
      O     M   1001.2;
      )     ;
      A     M   1208.0;
      A     M   1208.5;
      AN    M   1208.3;
      AN    M   1243.4;
      =     M   1243.5;
NETWORK
TITLE =
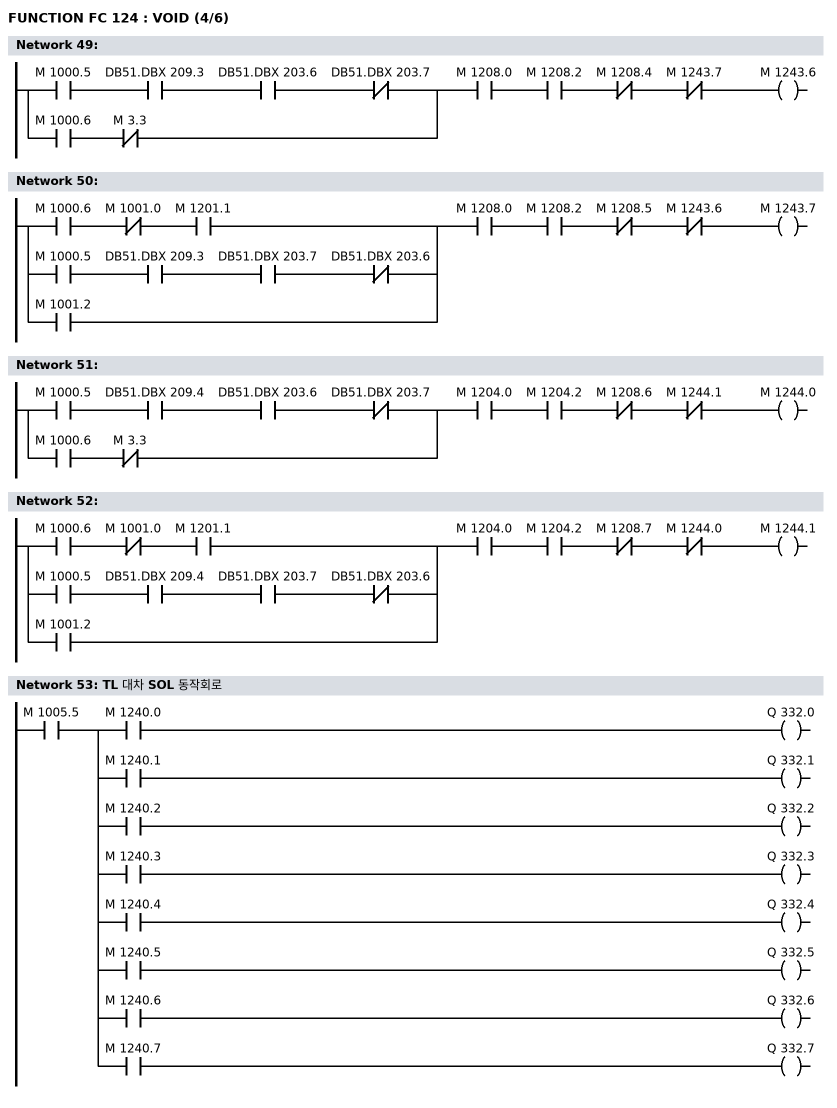

      A(    ;
      A     M   1000.5;
      A     DB51.DBX  209.3;
      A     DB51.DBX  203.6;
      AN    DB51.DBX  203.7;
      O     ;
      A     M   1000.6;
      AN    M      3.3;
      )     ;
      A     M   1208.0;
      A     M   1208.2;
      AN    M   1208.4;
      AN    M   1243.7;
      =     M   1243.6;
NETWORK
TITLE =

      A(    ;
      A     M   1000.6;
      AN    M   1001.0;
      A     M   1201.1;
      O     ;
      A     M   1000.5;
      A     DB51.DBX  209.3;
      A     DB51.DBX  203.7;
      AN    DB51.DBX  203.6;
      O     M   1001.2;
      )     ;
      A     M   1208.0;
      A     M   1208.2;
      AN    M   1208.5;
      AN    M   1243.6;
      =     M   1243.7;
NETWORK
TITLE =

      A(    ;
      A     M   1000.5;
      A     DB51.DBX  209.4;
      A     DB51.DBX  203.6;
      AN    DB51.DBX  203.7;
      O     ;
      A     M   1000.6;
      AN    M      3.3;
      )     ;
      A     M   1204.0;
      A     M   1204.2;
      AN    M   1208.6;
      AN    M   1244.1;
      =     M   1244.0;
NETWORK
TITLE =

      A(    ;
      A     M   1000.6;
      AN    M   1001.0;
      A     M   1201.1;
      O     ;
      A     M   1000.5;
      A     DB51.DBX  209.4;
      A     DB51.DBX  203.7;
      AN    DB51.DBX  203.6;
      O     M   1001.2;
      )     ;
      A     M   1204.0;
      A     M   1204.2;
      AN    M   1208.7;
      AN    M   1244.0;
      =     M   1244.1;
NETWORK
TITLE =TL 대차 SOL 동작회로

      A     M   1005.5;
      =     L      0.0;
      A     L      0.0;
      A     M   1240.0;
      =     Q    332.0;
      A     L      0.0;
      A     M   1240.1;
      =     Q    332.1;
      A     L      0.0;
      A     M   1240.2;
      =     Q    332.2;
      A     L      0.0;
      A     M   1240.3;
      =     Q    332.3;
      A     L      0.0;
      A     M   1240.4;
      =     Q    332.4;
      A     L      0.0;
      A     M   1240.5;
      =     Q    332.5;
      A     L      0.0;
      A     M   1240.6;
      =     Q    332.6;
      A     L      0.0;
      A     M   1240.7;
      =     Q    332.7;
NETWORK
TITLE =
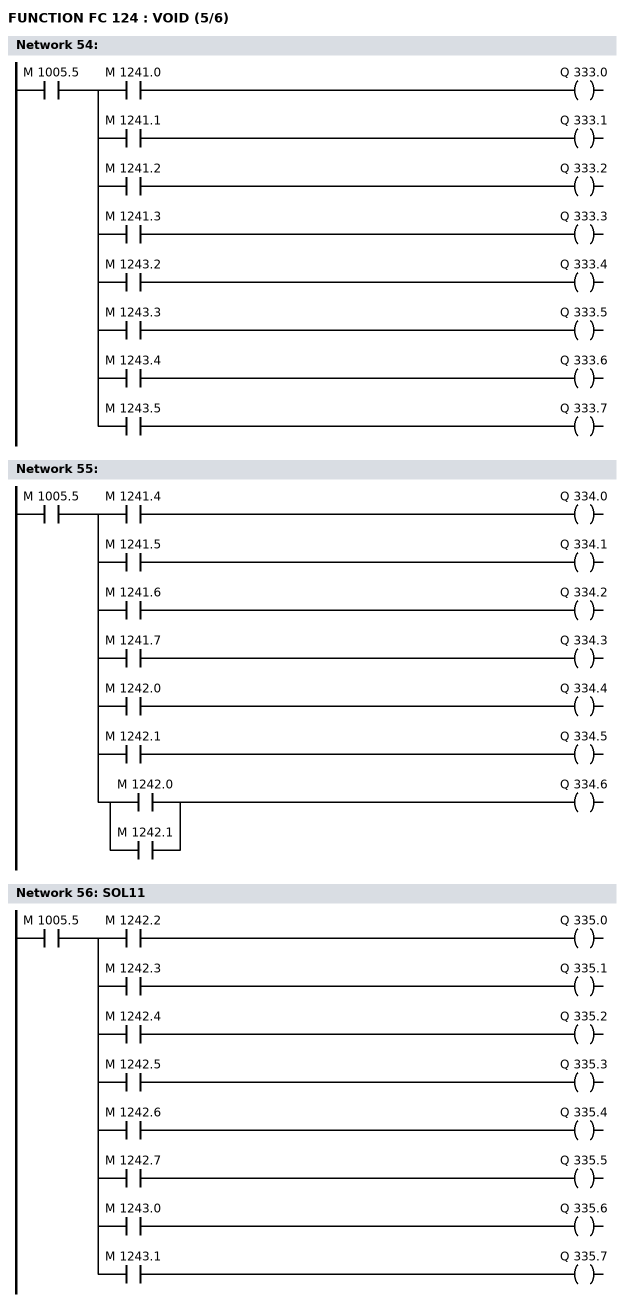

      A     M   1005.5;
      =     L      0.0;
      A     L      0.0;
      A     M   1241.0;
      =     Q    333.0;
      A     L      0.0;
      A     M   1241.1;
      =     Q    333.1;
      A     L      0.0;
      A     M   1241.2;
      =     Q    333.2;
      A     L      0.0;
      A     M   1241.3;
      =     Q    333.3;
      A     L      0.0;
      A     M   1243.2;
      =     Q    333.4;
      A     L      0.0;
      A     M   1243.3;
      =     Q    333.5;
      A     L      0.0;
      A     M   1243.4;
      =     Q    333.6;
      A     L      0.0;
      A     M   1243.5;
      =     Q    333.7;
NETWORK
TITLE =

      A     M   1005.5;
      =     L      0.0;
      A     L      0.0;
      A     M   1241.4;
      =     Q    334.0;
      A     L      0.0;
      A     M   1241.5;
      =     Q    334.1;
      A     L      0.0;
      A     M   1241.6;
      =     Q    334.2;
      A     L      0.0;
      A     M   1241.7;
      =     Q    334.3;
      A     L      0.0;
      A     M   1242.0;
      =     Q    334.4;
      A     L      0.0;
      A     M   1242.1;
      =     Q    334.5;
      A     L      0.0;
      A(    ;
      O     M   1242.0;
      O     M   1242.1;
      )     ;
      =     Q    334.6;
NETWORK
TITLE =SOL11

      A     M   1005.5;
      =     L      0.0;
      A     L      0.0;
      A     M   1242.2;
      =     Q    335.0;
      A     L      0.0;
      A     M   1242.3;
      =     Q    335.1;
      A     L      0.0;
      A     M   1242.4;
      =     Q    335.2;
      A     L      0.0;
      A     M   1242.5;
      =     Q    335.3;
      A     L      0.0;
      A     M   1242.6;
      =     Q    335.4;
      A     L      0.0;
      A     M   1242.7;
      =     Q    335.5;
      A     L      0.0;
      A     M   1243.0;
      =     Q    335.6;
      A     L      0.0;
      A     M   1243.1;
      =     Q    335.7;
NETWORK
TITLE =
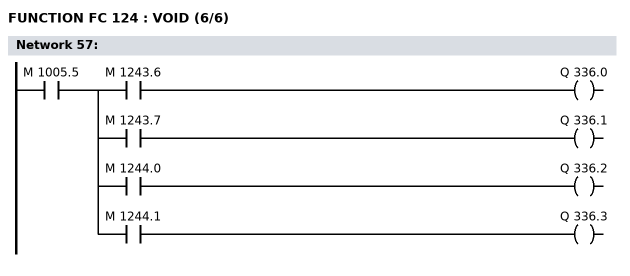

      A     M   1005.5;
      =     L      0.0;
      A     L      0.0;
      A     M   1243.6;
      =     Q    336.0;
      A     L      0.0;
      A     M   1243.7;
      =     Q    336.1;
      A     L      0.0;
      A     M   1244.0;
      =     Q    336.2;
      A     L      0.0;
      A     M   1244.1;
      =     Q    336.3;
END_FUNCTION

FUNCTION FC 125 : VOID
TITLE =
VERSION : 0.1

BEGIN
NETWORK
TITLE =
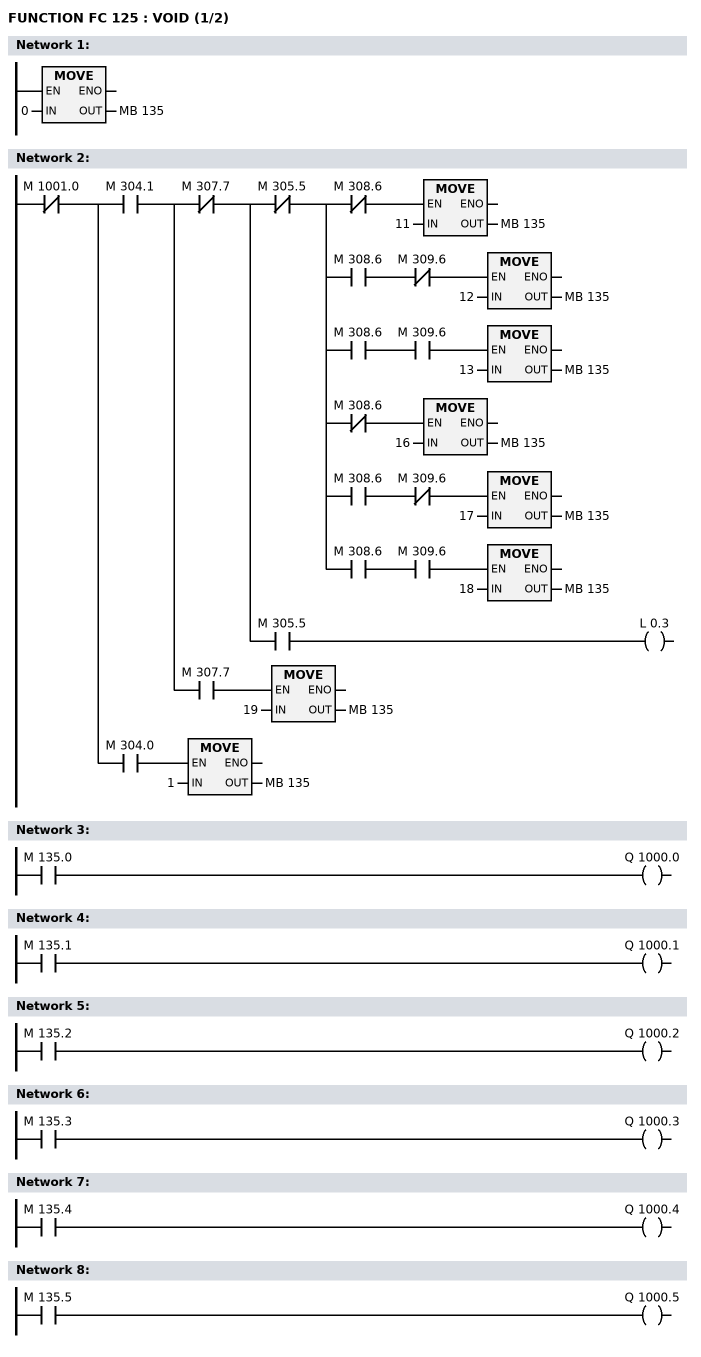

      L     0;
      T     MB   135;
      NOP   0;
NETWORK
TITLE =

      AN    M   1001.0;
      =     L      0.0;
      A     L      0.0;
      A     M    304.1;
      =     L      0.1;
      A     L      0.1;
      AN    M    307.7;
      =     L      0.2;
      A     L      0.2;
      AN    M    305.5;
      =     L      0.3;
      A     L      0.3;
      AN    M    308.6;
      JNB   _001;
      L     11;
      T     MB   135;
_001: NOP   0;
      A     L      0.3;
      A     M    308.6;
      AN    M    309.6;
      JNB   _002;
      L     12;
      T     MB   135;
_002: NOP   0;
      A     L      0.3;
      A     M    308.6;
      A     M    309.6;
      JNB   _003;
      L     13;
      T     MB   135;
_003: NOP   0;
      A     L      0.2;
      A     M    305.5;
      =     L      0.3;
      A     L      0.3;
      AN    M    308.6;
      JNB   _004;
      L     16;
      T     MB   135;
_004: NOP   0;
      A     L      0.3;
      A     M    308.6;
      AN    M    309.6;
      JNB   _005;
      L     17;
      T     MB   135;
_005: NOP   0;
      A     L      0.3;
      A     M    308.6;
      A     M    309.6;
      JNB   _006;
      L     18;
      T     MB   135;
_006: NOP   0;
      A     L      0.1;
      A     M    307.7;
      JNB   _007;
      L     19;
      T     MB   135;
_007: NOP   0;
      A     L      0.0;
      A     M    304.0;
      JNB   _008;
      L     1;
      T     MB   135;
_008: NOP   0;
NETWORK
TITLE =

      A     M    135.0;
      =     Q   1000.0;
NETWORK
TITLE =

      A     M    135.1;
      =     Q   1000.1;
NETWORK
TITLE =

      A     M    135.2;
      =     Q   1000.2;
NETWORK
TITLE =

      A     M    135.3;
      =     Q   1000.3;
NETWORK
TITLE =

      A     M    135.4;
      =     Q   1000.4;
NETWORK
TITLE =

      A     M    135.5;
      =     Q   1000.5;
NETWORK
TITLE =
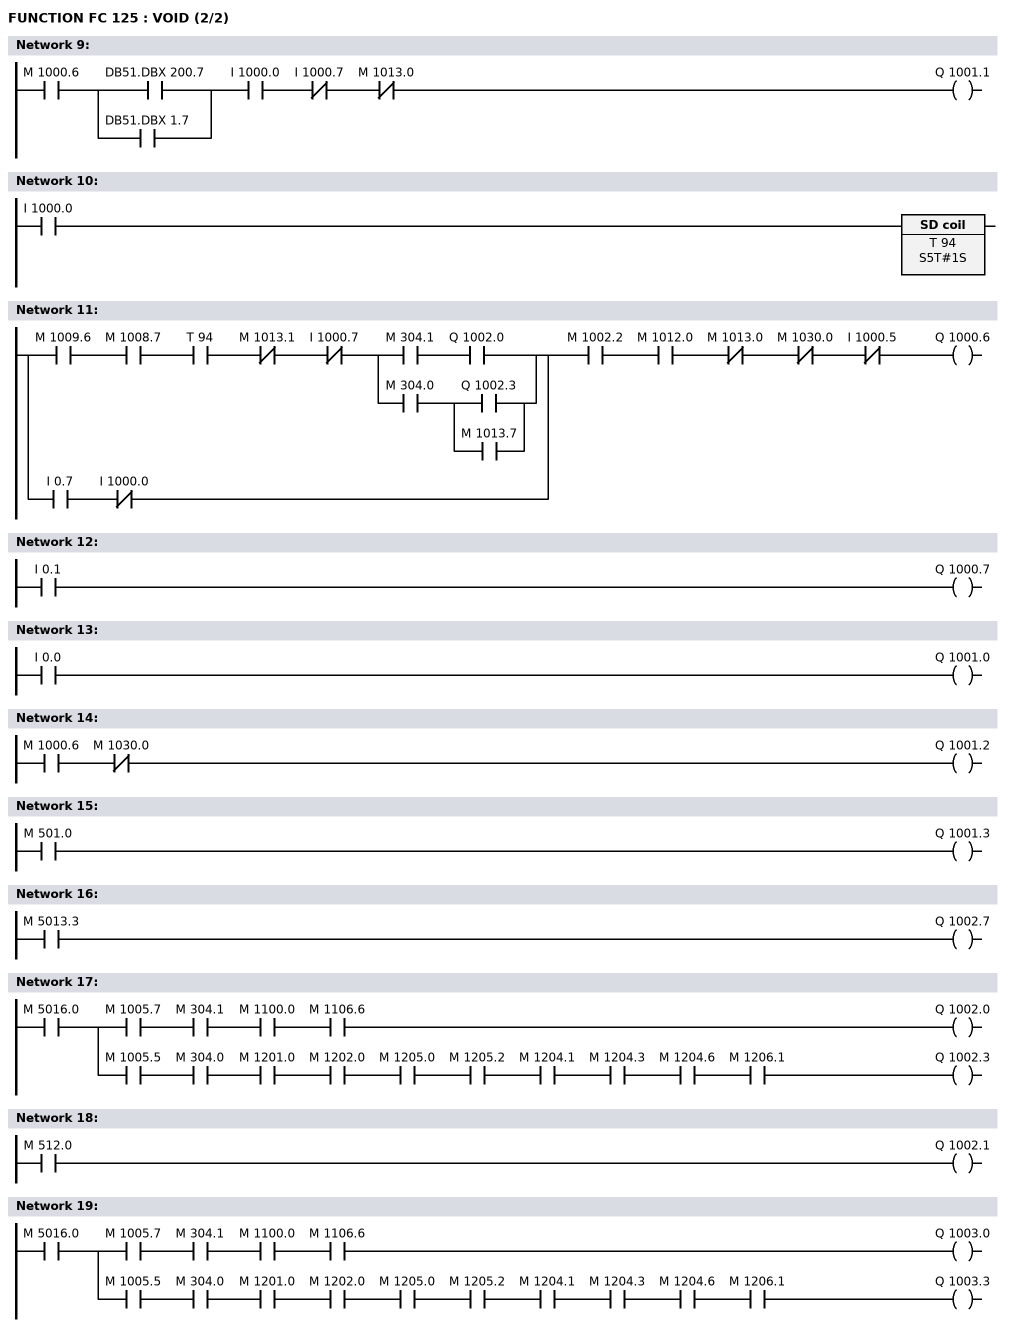

      A     M   1000.6;
      A(    ;
      O     DB51.DBX  200.7;
      O     DB51.DBX    1.7;
      )     ;
      A     I   1000.0;
      AN    I   1000.7;
      AN    M   1013.0;
      =     Q   1001.1;
NETWORK
TITLE =

      A     I   1000.0;
      L     S5T#1S;
      SD    T     94;
NETWORK
TITLE =

      A(    ;
      A     M   1009.6;
      A     M   1008.7;
      A     T     94;
      AN    M   1013.1;
      AN    I   1000.7;
      A(    ;
      A     M    304.1;
      A     Q   1002.0;
      O     ;
      A     M    304.0;
      A(    ;
      O     Q   1002.3;
      O     M   1013.7;
      )     ;
      )     ;
      O     ;
      A     I      0.7;
      AN    I   1000.0;
      )     ;
      A     M   1002.2;
      A     M   1012.0;
      AN    M   1013.0;
      AN    M   1030.0;
      AN    I   1000.5;
      =     Q   1000.6;
NETWORK
TITLE =

      A     I      0.1;
      =     Q   1000.7;
NETWORK
TITLE =

      A     I      0.0;
      =     Q   1001.0;
NETWORK
TITLE =

      A     M   1000.6;
      AN    M   1030.0;
      =     Q   1001.2;
NETWORK
TITLE =

      A     M    501.0;
      =     Q   1001.3;
NETWORK
TITLE =

      A     M   5013.3;
      =     Q   1002.7;
NETWORK
TITLE =

      A     M   5016.0;
      =     L      0.0;
      A     L      0.0;
      A     M   1005.7;
      A     M    304.1;
      A     M   1100.0;
      A     M   1106.6;
      =     Q   1002.0;
      A     L      0.0;
      A     M   1005.5;
      A     M    304.0;
      A     M   1201.0;
      A     M   1202.0;
      A     M   1205.0;
      A     M   1205.2;
      A     M   1204.1;
      A     M   1204.3;
      A     M   1204.6;
      A     M   1206.1;
      =     Q   1002.3;
NETWORK
TITLE =

      A     M    512.0;
      =     Q   1002.1;
NETWORK
TITLE =

      A     M   5016.0;
      =     L      0.0;
      A     L      0.0;
      A     M   1005.7;
      A     M    304.1;
      A     M   1100.0;
      A     M   1106.6;
      =     Q   1003.0;
      A     L      0.0;
      A     M   1005.5;
      A     M    304.0;
      A     M   1201.0;
      A     M   1202.0;
      A     M   1205.0;
      A     M   1205.2;
      A     M   1204.1;
      A     M   1204.3;
      A     M   1204.6;
      A     M   1206.1;
      =     Q   1003.3;
END_FUNCTION

FUNCTION_BLOCK FB 130
TITLE =
VERSION : 0.1


VAR
  S703_MODE : FB 402;
END_VAR
BEGIN
NETWORK
TITLE =
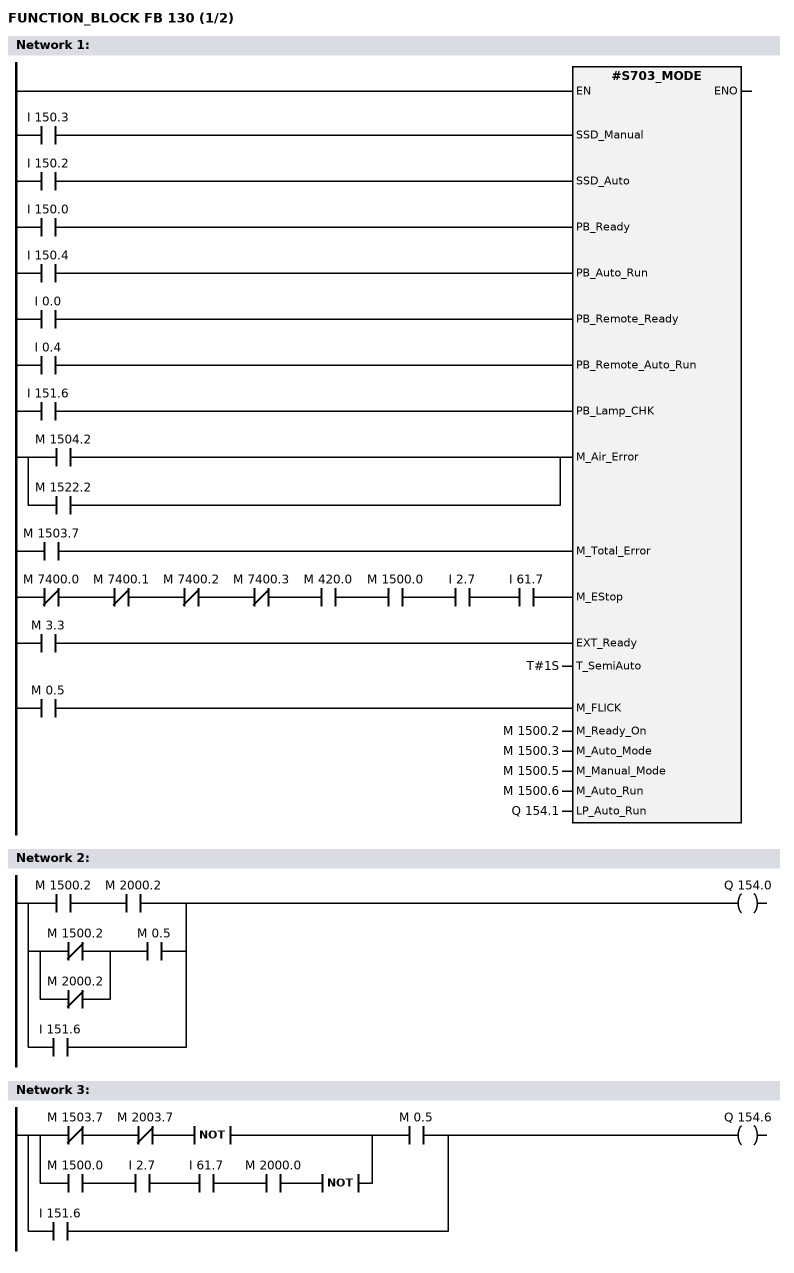

      A     I    150.3;
      =     L      0.0;
      BLD   103;
      A     I    150.2;
      =     L      0.1;
      BLD   103;
      A     I    150.0;
      =     L      0.2;
      BLD   103;
      A     I    150.4;
      =     L      0.3;
      BLD   103;
      A     I      0.0;
      =     L      0.4;
      BLD   103;
      A     I      0.4;
      =     L      0.5;
      BLD   103;
      A     I    151.6;
      =     L      0.6;
      BLD   103;
      A(    ;
      O     M   1504.2;
      O     M   1522.2;
      )     ;
      =     L      0.7;
      BLD   103;
      A     M   1503.7;
      =     L      1.1;
      BLD   103;
      AN    M   7400.0;
      AN    M   7400.1;
      AN    M   7400.2;
      AN    M   7400.3;
      A     M    420.0;
      A     M   1500.0;
      A     I      2.7;
      A     I     61.7;
      =     L      1.2;
      BLD   103;
      A     M      3.3;
      =     L      1.3;
      BLD   103;
      A     M      0.5;
      =     L      1.5;
      BLD   103;
      CALL #S703_MODE (
           SSD_Manual               := L      0.0,
           SSD_Auto                 := L      0.1,
           PB_Ready                 := L      0.2,
           PB_Auto_Run              := L      0.3,
           PB_Remote_Ready          := L      0.4,
           PB_Remote_Auto_Run       := L      0.5,
           PB_Lamp_CHK              := L      0.6,
           M_Air_Error              := L      0.7,
           M_Total_Error            := L      1.1,
           M_EStop                  := L      1.2,
           EXT_Ready                := L      1.3,
           T_SemiAuto               := T#1S,
           M_FLICK                  := L      1.5,
           M_Ready_On               := M   1500.2,
           M_Auto_Mode              := M   1500.3,
           M_Manual_Mode            := M   1500.5,
           M_Auto_Run               := M   1500.6,
           LP_Auto_Run              := Q    154.1);
      NOP   0;
NETWORK
TITLE =

      A     M   1500.2;
      A     M   2000.2;
      O     ;
      A(    ;
      ON    M   1500.2;
      ON    M   2000.2;
      )     ;
      A     M      0.5;
      O     I    151.6;
      =     Q    154.0;
NETWORK
TITLE =

      A(    ;
      AN    M   1503.7;
      AN    M   2003.7;
      NOT   ;
      O(    ;
      A     M   1500.0;
      A     I      2.7;
      A     I     61.7;
      A     M   2000.0;
      NOT   ;
      )     ;
      )     ;
      A     M      0.5;
      O     I    151.6;
      =     Q    154.6;
NETWORK
TITLE =
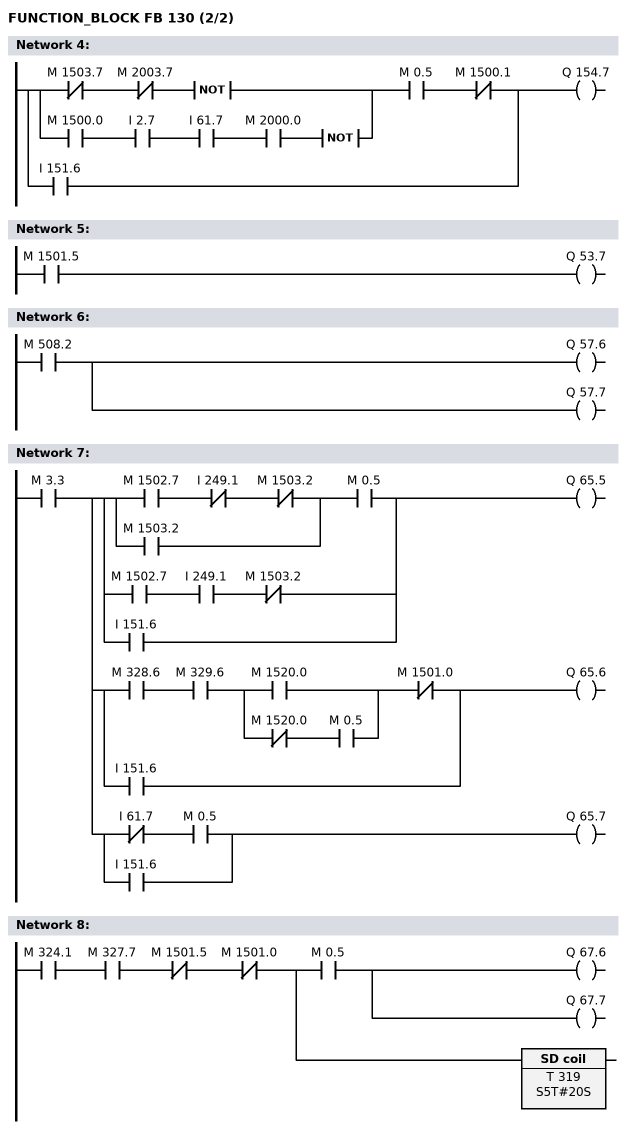

      A(    ;
      AN    M   1503.7;
      AN    M   2003.7;
      NOT   ;
      O(    ;
      A     M   1500.0;
      A     I      2.7;
      A     I     61.7;
      A     M   2000.0;
      NOT   ;
      )     ;
      )     ;
      A     M      0.5;
      AN    M   1500.1;
      O     I    151.6;
      =     Q    154.7;
NETWORK
TITLE =

      A     M   1501.5;
      =     Q     53.7;
NETWORK
TITLE =

      A     M    508.2;
      =     Q     57.6;
      =     Q     57.7;
NETWORK
TITLE =

      A     M      3.3;
      =     L      0.0;
      A     L      0.0;
      A(    ;
      A(    ;
      A     M   1502.7;
      AN    I    249.1;
      AN    M   1503.2;
      O     M   1503.2;
      )     ;
      A     M      0.5;
      O     ;
      A     M   1502.7;
      A     I    249.1;
      AN    M   1503.2;
      O     I    151.6;
      )     ;
      =     Q     65.5;
      A     L      0.0;
      A(    ;
      A     M    328.6;
      A     M    329.6;
      A(    ;
      O     M   1520.0;
      O     ;
      AN    M   1520.0;
      A     M      0.5;
      )     ;
      AN    M   1501.0;
      O     I    151.6;
      )     ;
      =     Q     65.6;
      A     L      0.0;
      A(    ;
      AN    I     61.7;
      A     M      0.5;
      O     I    151.6;
      )     ;
      =     Q     65.7;
NETWORK
TITLE =

      A     M    324.1;
      A     M    327.7;
      AN    M   1501.5;
      AN    M   1501.0;
      =     L      0.0;
      A     L      0.0;
      A     M      0.5;
      =     Q     67.6;
      =     Q     67.7;
      A     L      0.0;
      BLD   102;
      L     S5T#20S;
      SD    T    319;
END_FUNCTION_BLOCK

DATA_BLOCK DB 130
TITLE =
VERSION : 0.0

 FB 130
BEGIN
   S703_MODE.SSD_Manual := FALSE;
   S703_MODE.SSD_Auto := FALSE;
   S703_MODE.PB_Ready := FALSE;
   S703_MODE.PB_Auto_Run := FALSE;
   S703_MODE.PB_Remote_Ready := FALSE;
   S703_MODE.PB_Remote_Auto_Run := FALSE;
   S703_MODE.PB_Lamp_CHK := FALSE;
   S703_MODE.M_Air_Error := FALSE;
   S703_MODE.M_Water_Error := FALSE;
   S703_MODE.M_Total_Error := FALSE;
   S703_MODE.M_EStop := FALSE;
   S703_MODE.EXT_Ready := FALSE;
   S703_MODE.EXT_Auto := FALSE;
   S703_MODE.T_SemiAuto := T#0MS;
   S703_MODE.M_FLICK := FALSE;
   S703_MODE.M_Ready_On := FALSE;
   S703_MODE.M_Auto_Mode := FALSE;
   S703_MODE.M_SemiAuto_Mode := FALSE;
   S703_MODE.M_Manual_Mode := FALSE;
   S703_MODE.M_Auto_Run := FALSE;
   S703_MODE.LP_Ready_On := FALSE;
   S703_MODE.LP_Auto_Run := FALSE;
   S703_MODE.AUTO_MODE_DELAY.IN := FALSE;
   S703_MODE.AUTO_MODE_DELAY.PT := T#0MS;
   S703_MODE.AUTO_MODE_DELAY.Q := FALSE;
   S703_MODE.AUTO_MODE_DELAY.ET := T#0MS;
   S703_MODE.AUTO_MODE_DELAY.STATE := B#16#0;
   S703_MODE.AUTO_MODE_DELAY.STIME := T#0MS;
   S703_MODE.AUTO_MODE_DELAY.ATIME := T#0MS;
   S703_MODE.SEMI_AUTO_DELAY.IN := FALSE;
   S703_MODE.SEMI_AUTO_DELAY.PT := T#0MS;
   S703_MODE.SEMI_AUTO_DELAY.Q := FALSE;
   S703_MODE.SEMI_AUTO_DELAY.ET := T#0MS;
   S703_MODE.SEMI_AUTO_DELAY.STATE := B#16#0;
   S703_MODE.SEMI_AUTO_DELAY.STIME := T#0MS;
   S703_MODE.SEMI_AUTO_DELAY.ATIME := T#0MS;
   S703_MODE.MANUAL_DELAY.IN := FALSE;
   S703_MODE.MANUAL_DELAY.PT := T#0MS;
   S703_MODE.MANUAL_DELAY.Q := FALSE;
   S703_MODE.MANUAL_DELAY.ET := T#0MS;
   S703_MODE.MANUAL_DELAY.STATE := B#16#0;
   S703_MODE.MANUAL_DELAY.STIME := T#0MS;
   S703_MODE.MANUAL_DELAY.ATIME := T#0MS;
END_DATA_BLOCK

FUNCTION FC 130 : VOID
TITLE =
VERSION : 0.1

BEGIN
NETWORK
TITLE =
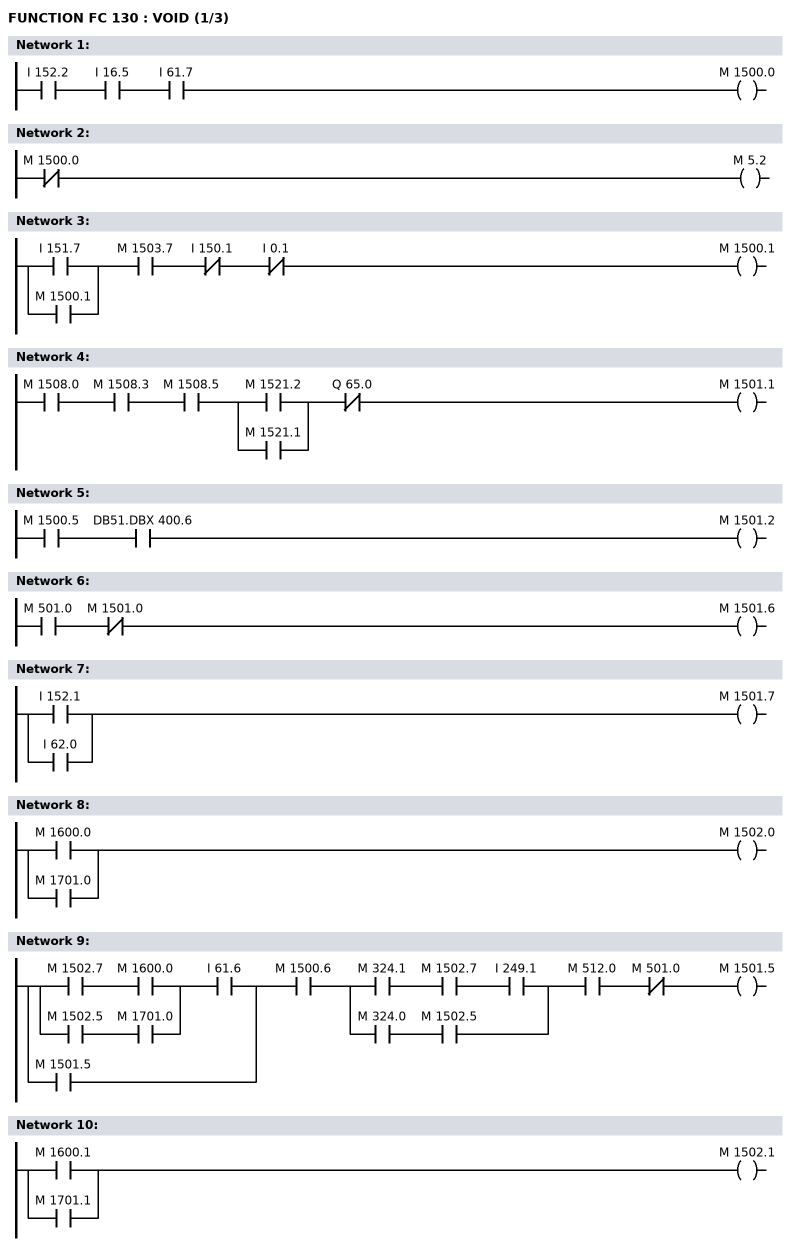

      A     I    152.2;
      A     I     16.5;
      A     I     61.7;
      =     M   1500.0;
NETWORK
TITLE =

      AN    M   1500.0;
      =     M      5.2;
NETWORK
TITLE =

      A(    ;
      O     I    151.7;
      O     M   1500.1;
      )     ;
      A     M   1503.7;
      AN    I    150.1;
      AN    I      0.1;
      =     M   1500.1;
NETWORK
TITLE =

      A     M   1508.0;
      A     M   1508.3;
      A     M   1508.5;
      A(    ;
      O     M   1521.2;
      O     M   1521.1;
      )     ;
      AN    Q     65.0;
      =     M   1501.1;
NETWORK
TITLE =

      A     M   1500.5;
      A     DB51.DBX  400.6;
      =     M   1501.2;
NETWORK
TITLE =

      A     M    501.0;
      AN    M   1501.0;
      =     M   1501.6;
NETWORK
TITLE =

      O     I    152.1;
      O     I     62.0;
      =     M   1501.7;
NETWORK
TITLE =

      O     M   1600.0;
      O     M   1701.0;
      =     M   1502.0;
NETWORK
TITLE =

      A(    ;
      A(    ;
      A     M   1502.7;
      A     M   1600.0;
      O     ;
      A     M   1502.5;
      A     M   1701.0;
      )     ;
      A     I     61.6;
      O     M   1501.5;
      )     ;
      A     M   1500.6;
      A(    ;
      A     M    324.1;
      A     M   1502.7;
      A     I    249.1;
      O     ;
      A     M    324.0;
      A     M   1502.5;
      )     ;
      A     M    512.0;
      AN    M    501.0;
      =     M   1501.5;
NETWORK
TITLE =

      O     M   1600.1;
      O     M   1701.1;
      =     M   1502.1;
NETWORK
TITLE =
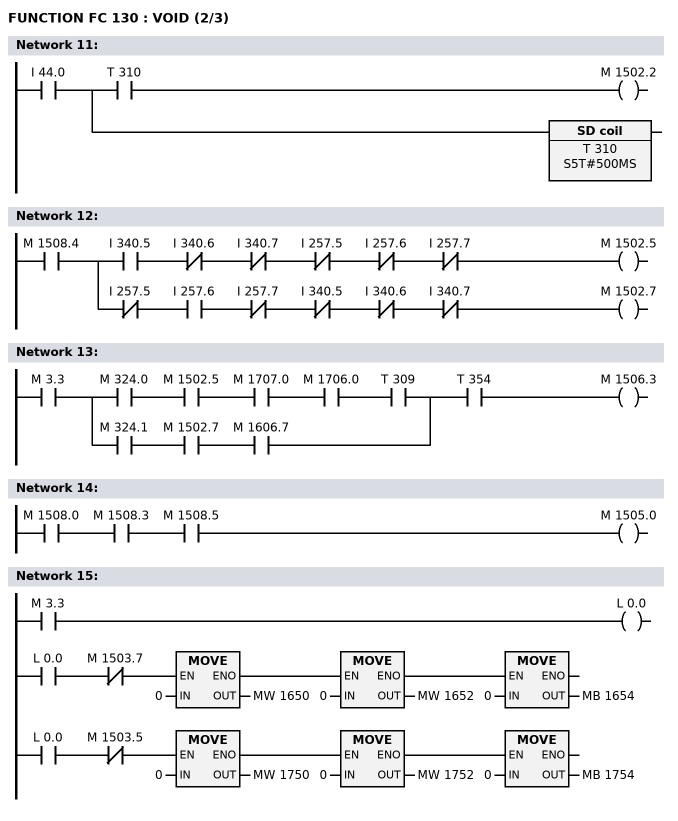

      A     I     44.0;
      =     L      0.0;
      A     L      0.0;
      A     T    310;
      =     M   1502.2;
      A     L      0.0;
      BLD   102;
      L     S5T#500MS;
      SD    T    310;
NETWORK
TITLE =

      A     M   1508.4;
      =     L      0.0;
      A     L      0.0;
      A     I    340.5;
      AN    I    340.6;
      AN    I    340.7;
      AN    I    257.5;
      AN    I    257.6;
      AN    I    257.7;
      =     M   1502.5;
      A     L      0.0;
      AN    I    257.5;
      A     I    257.6;
      AN    I    257.7;
      AN    I    340.5;
      AN    I    340.6;
      AN    I    340.7;
      =     M   1502.7;
NETWORK
TITLE =

      A     M      3.3;
      A(    ;
      A     M    324.0;
      A     M   1502.5;
      A     M   1707.0;
      A     M   1706.0;
      A     T    309;
      O     ;
      A     M    324.1;
      A     M   1502.7;
      A     M   1606.7;
      )     ;
      A     T    354;
      =     M   1506.3;
NETWORK
TITLE =

      A     M   1508.0;
      A     M   1508.3;
      A     M   1508.5;
      =     M   1505.0;
NETWORK
TITLE =

      A     M      3.3;
      =     L      0.0;
      A(    ;
      A(    ;
      A     L      0.0;
      AN    M   1503.7;
      JNB   _001;
      L     0;
      T     MW  1650;
      SET   ;
      SAVE  ;
      CLR   ;
_001: A     BR;
      )     ;
      JNB   _002;
      L     0;
      T     MW  1652;
      SET   ;
      SAVE  ;
      CLR   ;
_002: A     BR;
      )     ;
      JNB   _003;
      L     0;
      T     MB  1654;
_003: NOP   0;
      A(    ;
      A(    ;
      A     L      0.0;
      AN    M   1503.5;
      JNB   _004;
      L     0;
      T     MW  1750;
      SET   ;
      SAVE  ;
      CLR   ;
_004: A     BR;
      )     ;
      JNB   _005;
      L     0;
      T     MW  1752;
      SET   ;
      SAVE  ;
      CLR   ;
_005: A     BR;
      )     ;
      JNB   _006;
      L     0;
      T     MB  1754;
_006: NOP   0;
NETWORK
TITLE =
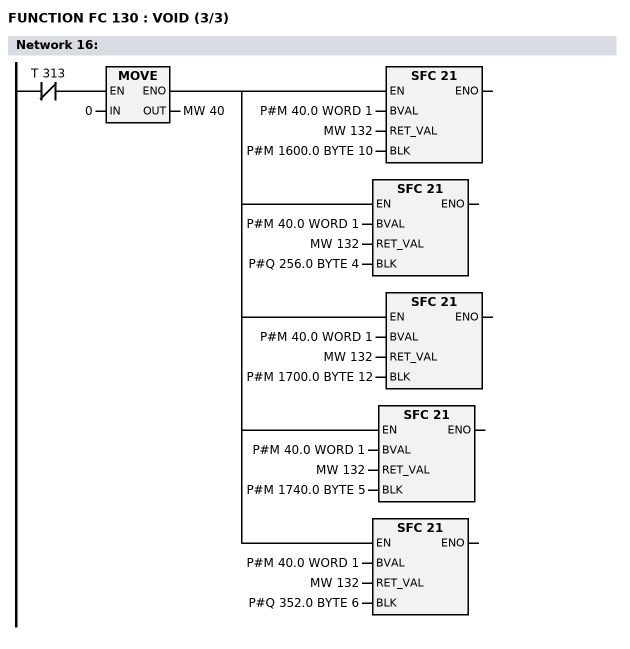

      AN    T    313;
      JNB   _007;
      L     0;
      T     MW    40;
      SET   ;
      SAVE  ;
      CLR   ;
_007: A     BR;
      =     L      0.0;
      A     L      0.0;
      JNB   _008;
      CALL SFC   21 (
           BVAL                     := P#M 40.0 WORD 1,
           RET_VAL                  := MW   132,
           BLK                      := P#M 1600.0 BYTE 10);
_008: NOP   0;
      A     L      0.0;
      JNB   _009;
      CALL SFC   21 (
           BVAL                     := P#M 40.0 WORD 1,
           RET_VAL                  := MW   132,
           BLK                      := P#Q 256.0 BYTE 4);
_009: NOP   0;
      A     L      0.0;
      JNB   _00a;
      CALL SFC   21 (
           BVAL                     := P#M 40.0 WORD 1,
           RET_VAL                  := MW   132,
           BLK                      := P#M 1700.0 BYTE 12);
_00a: NOP   0;
      A     L      0.0;
      JNB   _00b;
      CALL SFC   21 (
           BVAL                     := P#M 40.0 WORD 1,
           RET_VAL                  := MW   132,
           BLK                      := P#M 1740.0 BYTE 5);
_00b: NOP   0;
      A     L      0.0;
      JNB   _00c;
      CALL SFC   21 (
           BVAL                     := P#M 40.0 WORD 1,
           RET_VAL                  := MW   132,
           BLK                      := P#Q 352.0 BYTE 6);
_00c: NOP   0;
END_FUNCTION

FUNCTION_BLOCK FB 131
TITLE =
VERSION : 0.1


VAR
  S703_HOOK_PIN : FB 424;
  S703_DAECHA_LOCK : FB 424;
  S703_ELE : FB 424;
  S703_AIR_ELE : FB 424;
  S703_ROOF_RACK_A_R : FB 424;
  S703_ROOF_RACK_CLAMP : FB 424;
  S703_ROOF_RACK_GUN1_A_R : FB 424;
  S703_ROOF_RACK_GUN2_A_R : FB 424;
END_VAR
BEGIN
NETWORK
TITLE =
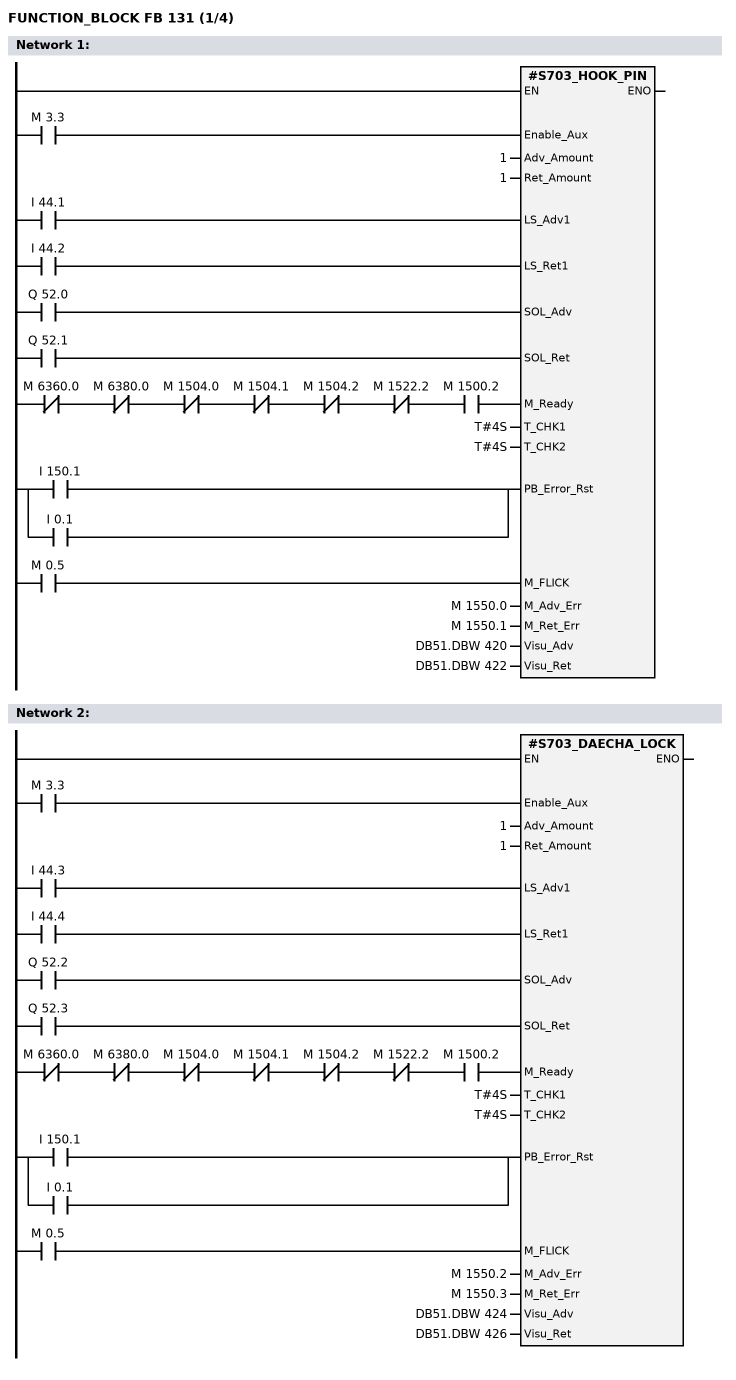

      A     M      3.3;
      =     L      0.0;
      BLD   103;
      A     I     44.1;
      =     L      0.1;
      BLD   103;
      A     I     44.2;
      =     L      0.2;
      BLD   103;
      A     Q     52.0;
      =     L      1.1;
      BLD   103;
      A     Q     52.1;
      =     L      1.2;
      BLD   103;
      AN    M   6360.0;
      AN    M   6380.0;
      AN    M   1504.0;
      AN    M   1504.1;
      AN    M   1504.2;
      AN    M   1522.2;
      A     M   1500.2;
      =     L      1.3;
      BLD   103;
      A(    ;
      O     I    150.1;
      O     I      0.1;
      )     ;
      =     L      1.5;
      BLD   103;
      A     M      0.5;
      =     L      1.6;
      BLD   103;
      CALL #S703_HOOK_PIN (
           Enable_Aux               := L      0.0,
           Adv_Amount               := 1,
           Ret_Amount               := 1,
           LS_Adv1                  := L      0.1,
           LS_Ret1                  := L      0.2,
           SOL_Adv                  := L      1.1,
           SOL_Ret                  := L      1.2,
           M_Ready                  := L      1.3,
           T_CHK1                   := T#4S,
           T_CHK2                   := T#4S,
           PB_Error_Rst             := L      1.5,
           M_FLICK                  := L      1.6,
           M_Adv_Err                := M   1550.0,
           M_Ret_Err                := M   1550.1,
           Visu_Adv                 := DB51.DBW  420,
           Visu_Ret                 := DB51.DBW  422);
      NOP   0;
NETWORK
TITLE =

      A     M      3.3;
      =     L      0.0;
      BLD   103;
      A     I     44.3;
      =     L      0.1;
      BLD   103;
      A     I     44.4;
      =     L      0.2;
      BLD   103;
      A     Q     52.2;
      =     L      1.1;
      BLD   103;
      A     Q     52.3;
      =     L      1.2;
      BLD   103;
      AN    M   6360.0;
      AN    M   6380.0;
      AN    M   1504.0;
      AN    M   1504.1;
      AN    M   1504.2;
      AN    M   1522.2;
      A     M   1500.2;
      =     L      1.3;
      BLD   103;
      A(    ;
      O     I    150.1;
      O     I      0.1;
      )     ;
      =     L      1.5;
      BLD   103;
      A     M      0.5;
      =     L      1.6;
      BLD   103;
      CALL #S703_DAECHA_LOCK (
           Enable_Aux               := L      0.0,
           Adv_Amount               := 1,
           Ret_Amount               := 1,
           LS_Adv1                  := L      0.1,
           LS_Ret1                  := L      0.2,
           SOL_Adv                  := L      1.1,
           SOL_Ret                  := L      1.2,
           M_Ready                  := L      1.3,
           T_CHK1                   := T#4S,
           T_CHK2                   := T#4S,
           PB_Error_Rst             := L      1.5,
           M_FLICK                  := L      1.6,
           M_Adv_Err                := M   1550.2,
           M_Ret_Err                := M   1550.3,
           Visu_Adv                 := DB51.DBW  424,
           Visu_Ret                 := DB51.DBW  426);
      NOP   0;
NETWORK
TITLE =
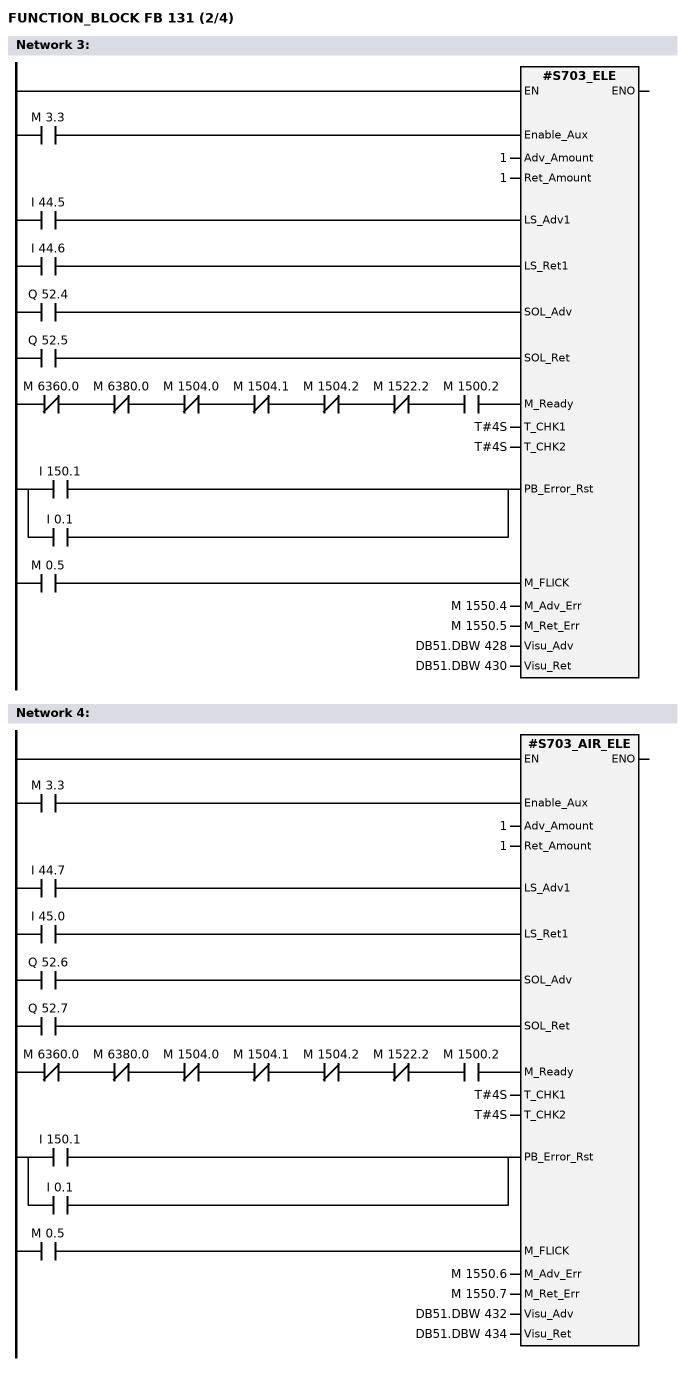

      A     M      3.3;
      =     L      0.0;
      BLD   103;
      A     I     44.5;
      =     L      0.1;
      BLD   103;
      A     I     44.6;
      =     L      0.2;
      BLD   103;
      A     Q     52.4;
      =     L      1.1;
      BLD   103;
      A     Q     52.5;
      =     L      1.2;
      BLD   103;
      AN    M   6360.0;
      AN    M   6380.0;
      AN    M   1504.0;
      AN    M   1504.1;
      AN    M   1504.2;
      AN    M   1522.2;
      A     M   1500.2;
      =     L      1.3;
      BLD   103;
      A(    ;
      O     I    150.1;
      O     I      0.1;
      )     ;
      =     L      1.5;
      BLD   103;
      A     M      0.5;
      =     L      1.6;
      BLD   103;
      CALL #S703_ELE (
           Enable_Aux               := L      0.0,
           Adv_Amount               := 1,
           Ret_Amount               := 1,
           LS_Adv1                  := L      0.1,
           LS_Ret1                  := L      0.2,
           SOL_Adv                  := L      1.1,
           SOL_Ret                  := L      1.2,
           M_Ready                  := L      1.3,
           T_CHK1                   := T#4S,
           T_CHK2                   := T#4S,
           PB_Error_Rst             := L      1.5,
           M_FLICK                  := L      1.6,
           M_Adv_Err                := M   1550.4,
           M_Ret_Err                := M   1550.5,
           Visu_Adv                 := DB51.DBW  428,
           Visu_Ret                 := DB51.DBW  430);
      NOP   0;
NETWORK
TITLE =

      A     M      3.3;
      =     L      0.0;
      BLD   103;
      A     I     44.7;
      =     L      0.1;
      BLD   103;
      A     I     45.0;
      =     L      0.2;
      BLD   103;
      A     Q     52.6;
      =     L      1.1;
      BLD   103;
      A     Q     52.7;
      =     L      1.2;
      BLD   103;
      AN    M   6360.0;
      AN    M   6380.0;
      AN    M   1504.0;
      AN    M   1504.1;
      AN    M   1504.2;
      AN    M   1522.2;
      A     M   1500.2;
      =     L      1.3;
      BLD   103;
      A(    ;
      O     I    150.1;
      O     I      0.1;
      )     ;
      =     L      1.5;
      BLD   103;
      A     M      0.5;
      =     L      1.6;
      BLD   103;
      CALL #S703_AIR_ELE (
           Enable_Aux               := L      0.0,
           Adv_Amount               := 1,
           Ret_Amount               := 1,
           LS_Adv1                  := L      0.1,
           LS_Ret1                  := L      0.2,
           SOL_Adv                  := L      1.1,
           SOL_Ret                  := L      1.2,
           M_Ready                  := L      1.3,
           T_CHK1                   := T#4S,
           T_CHK2                   := T#4S,
           PB_Error_Rst             := L      1.5,
           M_FLICK                  := L      1.6,
           M_Adv_Err                := M   1550.6,
           M_Ret_Err                := M   1550.7,
           Visu_Adv                 := DB51.DBW  432,
           Visu_Ret                 := DB51.DBW  434);
      NOP   0;
NETWORK
TITLE =

NETWORK
TITLE =
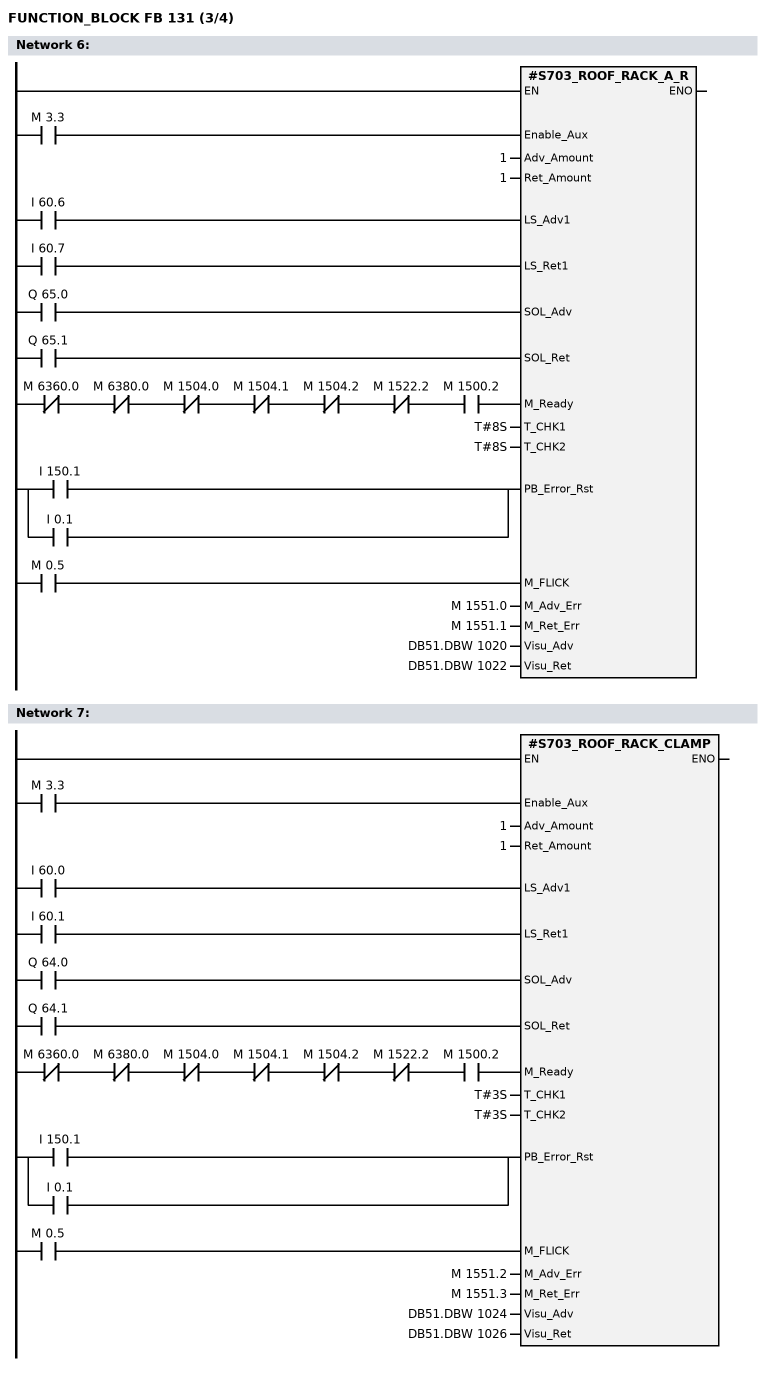

      A     M      3.3;
      =     L      0.0;
      BLD   103;
      A     I     60.6;
      =     L      0.1;
      BLD   103;
      A     I     60.7;
      =     L      0.2;
      BLD   103;
      A     Q     65.0;
      =     L      1.1;
      BLD   103;
      A     Q     65.1;
      =     L      1.2;
      BLD   103;
      AN    M   6360.0;
      AN    M   6380.0;
      AN    M   1504.0;
      AN    M   1504.1;
      AN    M   1504.2;
      AN    M   1522.2;
      A     M   1500.2;
      =     L      1.3;
      BLD   103;
      A(    ;
      O     I    150.1;
      O     I      0.1;
      )     ;
      =     L      1.5;
      BLD   103;
      A     M      0.5;
      =     L      1.6;
      BLD   103;
      CALL #S703_ROOF_RACK_A_R (
           Enable_Aux               := L      0.0,
           Adv_Amount               := 1,
           Ret_Amount               := 1,
           LS_Adv1                  := L      0.1,
           LS_Ret1                  := L      0.2,
           SOL_Adv                  := L      1.1,
           SOL_Ret                  := L      1.2,
           M_Ready                  := L      1.3,
           T_CHK1                   := T#8S,
           T_CHK2                   := T#8S,
           PB_Error_Rst             := L      1.5,
           M_FLICK                  := L      1.6,
           M_Adv_Err                := M   1551.0,
           M_Ret_Err                := M   1551.1,
           Visu_Adv                 := DB51.DBW 1020,
           Visu_Ret                 := DB51.DBW 1022);
      NOP   0;
NETWORK
TITLE =

      A     M      3.3;
      =     L      0.0;
      BLD   103;
      A     I     60.0;
      =     L      0.1;
      BLD   103;
      A     I     60.1;
      =     L      0.2;
      BLD   103;
      A     Q     64.0;
      =     L      1.1;
      BLD   103;
      A     Q     64.1;
      =     L      1.2;
      BLD   103;
      AN    M   6360.0;
      AN    M   6380.0;
      AN    M   1504.0;
      AN    M   1504.1;
      AN    M   1504.2;
      AN    M   1522.2;
      A     M   1500.2;
      =     L      1.3;
      BLD   103;
      A(    ;
      O     I    150.1;
      O     I      0.1;
      )     ;
      =     L      1.5;
      BLD   103;
      A     M      0.5;
      =     L      1.6;
      BLD   103;
      CALL #S703_ROOF_RACK_CLAMP (
           Enable_Aux               := L      0.0,
           Adv_Amount               := 1,
           Ret_Amount               := 1,
           LS_Adv1                  := L      0.1,
           LS_Ret1                  := L      0.2,
           SOL_Adv                  := L      1.1,
           SOL_Ret                  := L      1.2,
           M_Ready                  := L      1.3,
           T_CHK1                   := T#3S,
           T_CHK2                   := T#3S,
           PB_Error_Rst             := L      1.5,
           M_FLICK                  := L      1.6,
           M_Adv_Err                := M   1551.2,
           M_Ret_Err                := M   1551.3,
           Visu_Adv                 := DB51.DBW 1024,
           Visu_Ret                 := DB51.DBW 1026);
      NOP   0;
NETWORK
TITLE =
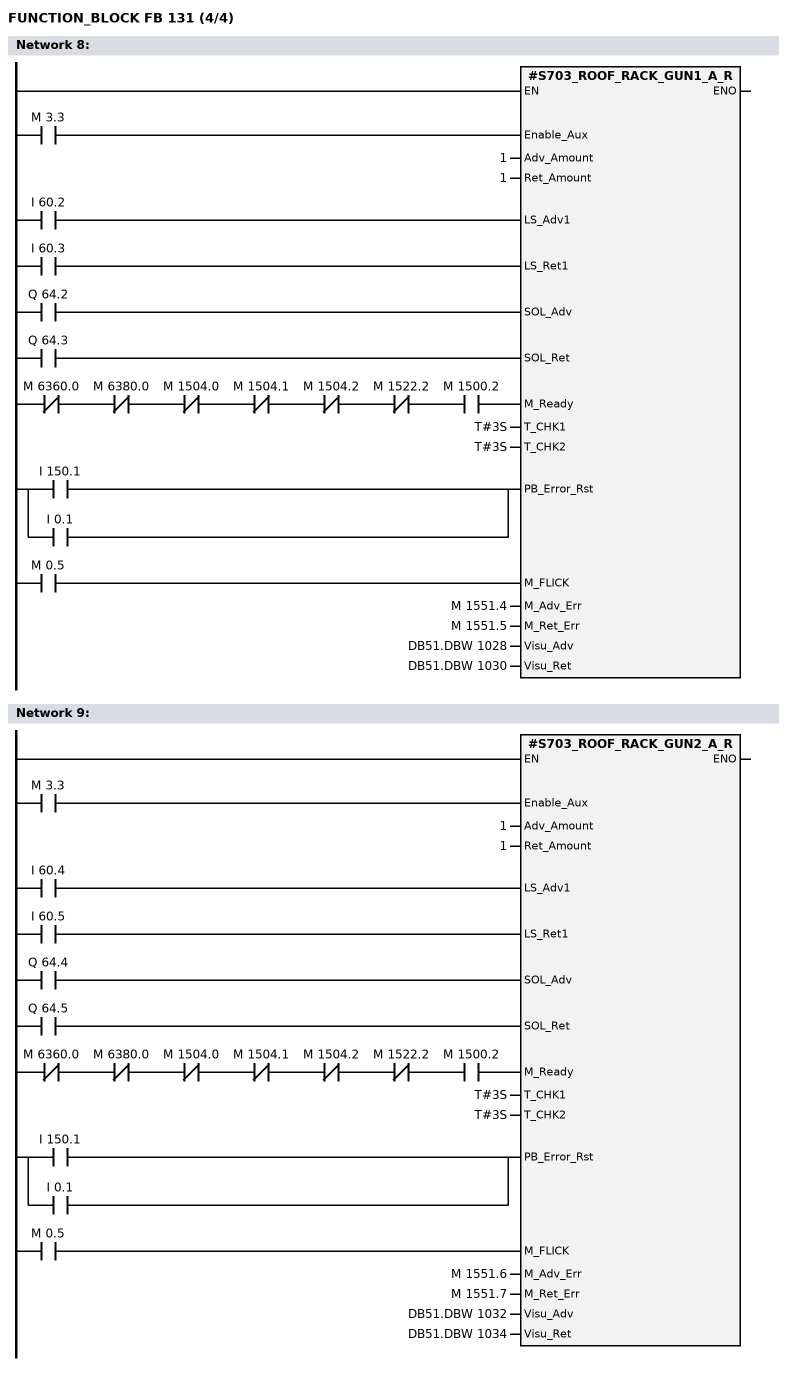

      A     M      3.3;
      =     L      0.0;
      BLD   103;
      A     I     60.2;
      =     L      0.1;
      BLD   103;
      A     I     60.3;
      =     L      0.2;
      BLD   103;
      A     Q     64.2;
      =     L      1.1;
      BLD   103;
      A     Q     64.3;
      =     L      1.2;
      BLD   103;
      AN    M   6360.0;
      AN    M   6380.0;
      AN    M   1504.0;
      AN    M   1504.1;
      AN    M   1504.2;
      AN    M   1522.2;
      A     M   1500.2;
      =     L      1.3;
      BLD   103;
      A(    ;
      O     I    150.1;
      O     I      0.1;
      )     ;
      =     L      1.5;
      BLD   103;
      A     M      0.5;
      =     L      1.6;
      BLD   103;
      CALL #S703_ROOF_RACK_GUN1_A_R (
           Enable_Aux               := L      0.0,
           Adv_Amount               := 1,
           Ret_Amount               := 1,
           LS_Adv1                  := L      0.1,
           LS_Ret1                  := L      0.2,
           SOL_Adv                  := L      1.1,
           SOL_Ret                  := L      1.2,
           M_Ready                  := L      1.3,
           T_CHK1                   := T#3S,
           T_CHK2                   := T#3S,
           PB_Error_Rst             := L      1.5,
           M_FLICK                  := L      1.6,
           M_Adv_Err                := M   1551.4,
           M_Ret_Err                := M   1551.5,
           Visu_Adv                 := DB51.DBW 1028,
           Visu_Ret                 := DB51.DBW 1030);
      NOP   0;
NETWORK
TITLE =

      A     M      3.3;
      =     L      0.0;
      BLD   103;
      A     I     60.4;
      =     L      0.1;
      BLD   103;
      A     I     60.5;
      =     L      0.2;
      BLD   103;
      A     Q     64.4;
      =     L      1.1;
      BLD   103;
      A     Q     64.5;
      =     L      1.2;
      BLD   103;
      AN    M   6360.0;
      AN    M   6380.0;
      AN    M   1504.0;
      AN    M   1504.1;
      AN    M   1504.2;
      AN    M   1522.2;
      A     M   1500.2;
      =     L      1.3;
      BLD   103;
      A(    ;
      O     I    150.1;
      O     I      0.1;
      )     ;
      =     L      1.5;
      BLD   103;
      A     M      0.5;
      =     L      1.6;
      BLD   103;
      CALL #S703_ROOF_RACK_GUN2_A_R (
           Enable_Aux               := L      0.0,
           Adv_Amount               := 1,
           Ret_Amount               := 1,
           LS_Adv1                  := L      0.1,
           LS_Ret1                  := L      0.2,
           SOL_Adv                  := L      1.1,
           SOL_Ret                  := L      1.2,
           M_Ready                  := L      1.3,
           T_CHK1                   := T#3S,
           T_CHK2                   := T#3S,
           PB_Error_Rst             := L      1.5,
           M_FLICK                  := L      1.6,
           M_Adv_Err                := M   1551.6,
           M_Ret_Err                := M   1551.7,
           Visu_Adv                 := DB51.DBW 1032,
           Visu_Ret                 := DB51.DBW 1034);
      NOP   0;
END_FUNCTION_BLOCK

DATA_BLOCK DB 131
TITLE =
VERSION : 0.0

 FB 131
BEGIN
   S703_HOOK_PIN.Enable_Aux := FALSE;
   S703_HOOK_PIN.Adv_Amount := 0;
   S703_HOOK_PIN.Ret_Amount := 0;
   S703_HOOK_PIN.LS_Adv1 := FALSE;
   S703_HOOK_PIN.LS_Ret1 := FALSE;
   S703_HOOK_PIN.LS_Adv2 := FALSE;
   S703_HOOK_PIN.LS_Ret2 := FALSE;
   S703_HOOK_PIN.LS_Adv3 := FALSE;
   S703_HOOK_PIN.LS_Ret3 := FALSE;
   S703_HOOK_PIN.LS_Adv4 := FALSE;
   S703_HOOK_PIN.LS_Ret4 := FALSE;
   S703_HOOK_PIN.SOL_Adv := FALSE;
   S703_HOOK_PIN.SOL_Ret := FALSE;
   S703_HOOK_PIN.M_Ready := FALSE;
   S703_HOOK_PIN.T_CHK1 := T#0MS;
   S703_HOOK_PIN.T_CHK2 := T#0MS;
   S703_HOOK_PIN.PB_Lamp_CHK := FALSE;
   S703_HOOK_PIN.PB_Error_Rst := FALSE;
   S703_HOOK_PIN.M_FLICK := FALSE;
   S703_HOOK_PIN.M_Adv_Err := FALSE;
   S703_HOOK_PIN.M_Ret_Err := FALSE;
   S703_HOOK_PIN.LP_Adv := FALSE;
   S703_HOOK_PIN.LP_Ret := FALSE;
   S703_HOOK_PIN.Visu_Adv := W#16#0;
   S703_HOOK_PIN.Visu_Ret := W#16#0;
   S703_HOOK_PIN.Error_T1.IN := FALSE;
   S703_HOOK_PIN.Error_T1.PT := T#0MS;
   S703_HOOK_PIN.Error_T1.Q := FALSE;
   S703_HOOK_PIN.Error_T1.ET := T#0MS;
   S703_HOOK_PIN.Error_T1.STATE := B#16#0;
   S703_HOOK_PIN.Error_T1.STIME := T#0MS;
   S703_HOOK_PIN.Error_T1.ATIME := T#0MS;
   S703_HOOK_PIN.Error_T2.IN := FALSE;
   S703_HOOK_PIN.Error_T2.PT := T#0MS;
   S703_HOOK_PIN.Error_T2.Q := FALSE;
   S703_HOOK_PIN.Error_T2.ET := T#0MS;
   S703_HOOK_PIN.Error_T2.STATE := B#16#0;
   S703_HOOK_PIN.Error_T2.STIME := T#0MS;
   S703_HOOK_PIN.Error_T2.ATIME := T#0MS;
   S703_HOOK_PIN.CHK_Aux1 := FALSE;
   S703_HOOK_PIN.CHK_Aux2 := FALSE;
   S703_HOOK_PIN.Error_T1_DN := FALSE;
   S703_HOOK_PIN.Error_T2_DN := FALSE;
   S703_HOOK_PIN.Adv_Memo := FALSE;
   S703_HOOK_PIN.Visu_Adv_Arr[0] := FALSE;
   S703_HOOK_PIN.Visu_Adv_Arr[1] := FALSE;
   S703_HOOK_PIN.Visu_Adv_Arr[2] := FALSE;
   S703_HOOK_PIN.Visu_Adv_Arr[3] := FALSE;
   S703_HOOK_PIN.Visu_Adv_Arr[4] := FALSE;
   S703_HOOK_PIN.Visu_Adv_Arr[5] := FALSE;
   S703_HOOK_PIN.Visu_Adv_Arr[6] := FALSE;
   S703_HOOK_PIN.Visu_Adv_Arr[7] := FALSE;
   S703_HOOK_PIN.Visu_Adv_Arr[8] := FALSE;
   S703_HOOK_PIN.Visu_Adv_Arr[9] := FALSE;
   S703_HOOK_PIN.Visu_Adv_Arr[10] := FALSE;
   S703_HOOK_PIN.Visu_Adv_Arr[11] := FALSE;
   S703_HOOK_PIN.Visu_Adv_Arr[12] := FALSE;
   S703_HOOK_PIN.Visu_Adv_Arr[13] := FALSE;
   S703_HOOK_PIN.Visu_Adv_Arr[14] := FALSE;
   S703_HOOK_PIN.Visu_Adv_Arr[15] := FALSE;
   S703_HOOK_PIN.Visu_Ret_Arr[0] := FALSE;
   S703_HOOK_PIN.Visu_Ret_Arr[1] := FALSE;
   S703_HOOK_PIN.Visu_Ret_Arr[2] := FALSE;
   S703_HOOK_PIN.Visu_Ret_Arr[3] := FALSE;
   S703_HOOK_PIN.Visu_Ret_Arr[4] := FALSE;
   S703_HOOK_PIN.Visu_Ret_Arr[5] := FALSE;
   S703_HOOK_PIN.Visu_Ret_Arr[6] := FALSE;
   S703_HOOK_PIN.Visu_Ret_Arr[7] := FALSE;
   S703_HOOK_PIN.Visu_Ret_Arr[8] := FALSE;
   S703_HOOK_PIN.Visu_Ret_Arr[9] := FALSE;
   S703_HOOK_PIN.Visu_Ret_Arr[10] := FALSE;
   S703_HOOK_PIN.Visu_Ret_Arr[11] := FALSE;
   S703_HOOK_PIN.Visu_Ret_Arr[12] := FALSE;
   S703_HOOK_PIN.Visu_Ret_Arr[13] := FALSE;
   S703_HOOK_PIN.Visu_Ret_Arr[14] := FALSE;
   S703_HOOK_PIN.Visu_Ret_Arr[15] := FALSE;
   S703_HOOK_PIN.BLK_Move_Ret := 0;
   S703_HOOK_PIN.Enable := FALSE;
   S703_HOOK_PIN.Adv_End := FALSE;
   S703_HOOK_PIN.Ret_End := FALSE;
   S703_DAECHA_LOCK.Enable_Aux := FALSE;
   S703_DAECHA_LOCK.Adv_Amount := 0;
   S703_DAECHA_LOCK.Ret_Amount := 0;
   S703_DAECHA_LOCK.LS_Adv1 := FALSE;
   S703_DAECHA_LOCK.LS_Ret1 := FALSE;
   S703_DAECHA_LOCK.LS_Adv2 := FALSE;
   S703_DAECHA_LOCK.LS_Ret2 := FALSE;
   S703_DAECHA_LOCK.LS_Adv3 := FALSE;
   S703_DAECHA_LOCK.LS_Ret3 := FALSE;
   S703_DAECHA_LOCK.LS_Adv4 := FALSE;
   S703_DAECHA_LOCK.LS_Ret4 := FALSE;
   S703_DAECHA_LOCK.SOL_Adv := FALSE;
   S703_DAECHA_LOCK.SOL_Ret := FALSE;
   S703_DAECHA_LOCK.M_Ready := FALSE;
   S703_DAECHA_LOCK.T_CHK1 := T#0MS;
   S703_DAECHA_LOCK.T_CHK2 := T#0MS;
   S703_DAECHA_LOCK.PB_Lamp_CHK := FALSE;
   S703_DAECHA_LOCK.PB_Error_Rst := FALSE;
   S703_DAECHA_LOCK.M_FLICK := FALSE;
   S703_DAECHA_LOCK.M_Adv_Err := FALSE;
   S703_DAECHA_LOCK.M_Ret_Err := FALSE;
   S703_DAECHA_LOCK.LP_Adv := FALSE;
   S703_DAECHA_LOCK.LP_Ret := FALSE;
   S703_DAECHA_LOCK.Visu_Adv := W#16#0;
   S703_DAECHA_LOCK.Visu_Ret := W#16#0;
   S703_DAECHA_LOCK.Error_T1.IN := FALSE;
   S703_DAECHA_LOCK.Error_T1.PT := T#0MS;
   S703_DAECHA_LOCK.Error_T1.Q := FALSE;
   S703_DAECHA_LOCK.Error_T1.ET := T#0MS;
   S703_DAECHA_LOCK.Error_T1.STATE := B#16#0;
   S703_DAECHA_LOCK.Error_T1.STIME := T#0MS;
   S703_DAECHA_LOCK.Error_T1.ATIME := T#0MS;
   S703_DAECHA_LOCK.Error_T2.IN := FALSE;
   S703_DAECHA_LOCK.Error_T2.PT := T#0MS;
   S703_DAECHA_LOCK.Error_T2.Q := FALSE;
   S703_DAECHA_LOCK.Error_T2.ET := T#0MS;
   S703_DAECHA_LOCK.Error_T2.STATE := B#16#0;
   S703_DAECHA_LOCK.Error_T2.STIME := T#0MS;
   S703_DAECHA_LOCK.Error_T2.ATIME := T#0MS;
   S703_DAECHA_LOCK.CHK_Aux1 := FALSE;
   S703_DAECHA_LOCK.CHK_Aux2 := FALSE;
   S703_DAECHA_LOCK.Error_T1_DN := FALSE;
   S703_DAECHA_LOCK.Error_T2_DN := FALSE;
   S703_DAECHA_LOCK.Adv_Memo := FALSE;
   S703_DAECHA_LOCK.Visu_Adv_Arr[0] := FALSE;
   S703_DAECHA_LOCK.Visu_Adv_Arr[1] := FALSE;
   S703_DAECHA_LOCK.Visu_Adv_Arr[2] := FALSE;
   S703_DAECHA_LOCK.Visu_Adv_Arr[3] := FALSE;
   S703_DAECHA_LOCK.Visu_Adv_Arr[4] := FALSE;
   S703_DAECHA_LOCK.Visu_Adv_Arr[5] := FALSE;
   S703_DAECHA_LOCK.Visu_Adv_Arr[6] := FALSE;
   S703_DAECHA_LOCK.Visu_Adv_Arr[7] := FALSE;
   S703_DAECHA_LOCK.Visu_Adv_Arr[8] := FALSE;
   S703_DAECHA_LOCK.Visu_Adv_Arr[9] := FALSE;
   S703_DAECHA_LOCK.Visu_Adv_Arr[10] := FALSE;
   S703_DAECHA_LOCK.Visu_Adv_Arr[11] := FALSE;
   S703_DAECHA_LOCK.Visu_Adv_Arr[12] := FALSE;
   S703_DAECHA_LOCK.Visu_Adv_Arr[13] := FALSE;
   S703_DAECHA_LOCK.Visu_Adv_Arr[14] := FALSE;
   S703_DAECHA_LOCK.Visu_Adv_Arr[15] := FALSE;
   S703_DAECHA_LOCK.Visu_Ret_Arr[0] := FALSE;
   S703_DAECHA_LOCK.Visu_Ret_Arr[1] := FALSE;
   S703_DAECHA_LOCK.Visu_Ret_Arr[2] := FALSE;
   S703_DAECHA_LOCK.Visu_Ret_Arr[3] := FALSE;
   S703_DAECHA_LOCK.Visu_Ret_Arr[4] := FALSE;
   S703_DAECHA_LOCK.Visu_Ret_Arr[5] := FALSE;
   S703_DAECHA_LOCK.Visu_Ret_Arr[6] := FALSE;
   S703_DAECHA_LOCK.Visu_Ret_Arr[7] := FALSE;
   S703_DAECHA_LOCK.Visu_Ret_Arr[8] := FALSE;
   S703_DAECHA_LOCK.Visu_Ret_Arr[9] := FALSE;
   S703_DAECHA_LOCK.Visu_Ret_Arr[10] := FALSE;
   S703_DAECHA_LOCK.Visu_Ret_Arr[11] := FALSE;
   S703_DAECHA_LOCK.Visu_Ret_Arr[12] := FALSE;
   S703_DAECHA_LOCK.Visu_Ret_Arr[13] := FALSE;
   S703_DAECHA_LOCK.Visu_Ret_Arr[14] := FALSE;
   S703_DAECHA_LOCK.Visu_Ret_Arr[15] := FALSE;
   S703_DAECHA_LOCK.BLK_Move_Ret := 0;
   S703_DAECHA_LOCK.Enable := FALSE;
   S703_DAECHA_LOCK.Adv_End := FALSE;
   S703_DAECHA_LOCK.Ret_End := FALSE;
   S703_ELE.Enable_Aux := FALSE;
   S703_ELE.Adv_Amount := 0;
   S703_ELE.Ret_Amount := 0;
   S703_ELE.LS_Adv1 := FALSE;
   S703_ELE.LS_Ret1 := FALSE;
   S703_ELE.LS_Adv2 := FALSE;
   S703_ELE.LS_Ret2 := FALSE;
   S703_ELE.LS_Adv3 := FALSE;
   S703_ELE.LS_Ret3 := FALSE;
   S703_ELE.LS_Adv4 := FALSE;
   S703_ELE.LS_Ret4 := FALSE;
   S703_ELE.SOL_Adv := FALSE;
   S703_ELE.SOL_Ret := FALSE;
   S703_ELE.M_Ready := FALSE;
   S703_ELE.T_CHK1 := T#0MS;
   S703_ELE.T_CHK2 := T#0MS;
   S703_ELE.PB_Lamp_CHK := FALSE;
   S703_ELE.PB_Error_Rst := FALSE;
   S703_ELE.M_FLICK := FALSE;
   S703_ELE.M_Adv_Err := FALSE;
   S703_ELE.M_Ret_Err := FALSE;
   S703_ELE.LP_Adv := FALSE;
   S703_ELE.LP_Ret := FALSE;
   S703_ELE.Visu_Adv := W#16#0;
   S703_ELE.Visu_Ret := W#16#0;
   S703_ELE.Error_T1.IN := FALSE;
   S703_ELE.Error_T1.PT := T#0MS;
   S703_ELE.Error_T1.Q := FALSE;
   S703_ELE.Error_T1.ET := T#0MS;
   S703_ELE.Error_T1.STATE := B#16#0;
   S703_ELE.Error_T1.STIME := T#0MS;
   S703_ELE.Error_T1.ATIME := T#0MS;
   S703_ELE.Error_T2.IN := FALSE;
   S703_ELE.Error_T2.PT := T#0MS;
   S703_ELE.Error_T2.Q := FALSE;
   S703_ELE.Error_T2.ET := T#0MS;
   S703_ELE.Error_T2.STATE := B#16#0;
   S703_ELE.Error_T2.STIME := T#0MS;
   S703_ELE.Error_T2.ATIME := T#0MS;
   S703_ELE.CHK_Aux1 := FALSE;
   S703_ELE.CHK_Aux2 := FALSE;
   S703_ELE.Error_T1_DN := FALSE;
   S703_ELE.Error_T2_DN := FALSE;
   S703_ELE.Adv_Memo := FALSE;
   S703_ELE.Visu_Adv_Arr[0] := FALSE;
   S703_ELE.Visu_Adv_Arr[1] := FALSE;
   S703_ELE.Visu_Adv_Arr[2] := FALSE;
   S703_ELE.Visu_Adv_Arr[3] := FALSE;
   S703_ELE.Visu_Adv_Arr[4] := FALSE;
   S703_ELE.Visu_Adv_Arr[5] := FALSE;
   S703_ELE.Visu_Adv_Arr[6] := FALSE;
   S703_ELE.Visu_Adv_Arr[7] := FALSE;
   S703_ELE.Visu_Adv_Arr[8] := FALSE;
   S703_ELE.Visu_Adv_Arr[9] := FALSE;
   S703_ELE.Visu_Adv_Arr[10] := FALSE;
   S703_ELE.Visu_Adv_Arr[11] := FALSE;
   S703_ELE.Visu_Adv_Arr[12] := FALSE;
   S703_ELE.Visu_Adv_Arr[13] := FALSE;
   S703_ELE.Visu_Adv_Arr[14] := FALSE;
   S703_ELE.Visu_Adv_Arr[15] := FALSE;
   S703_ELE.Visu_Ret_Arr[0] := FALSE;
   S703_ELE.Visu_Ret_Arr[1] := FALSE;
   S703_ELE.Visu_Ret_Arr[2] := FALSE;
   S703_ELE.Visu_Ret_Arr[3] := FALSE;
   S703_ELE.Visu_Ret_Arr[4] := FALSE;
   S703_ELE.Visu_Ret_Arr[5] := FALSE;
   S703_ELE.Visu_Ret_Arr[6] := FALSE;
   S703_ELE.Visu_Ret_Arr[7] := FALSE;
   S703_ELE.Visu_Ret_Arr[8] := FALSE;
   S703_ELE.Visu_Ret_Arr[9] := FALSE;
   S703_ELE.Visu_Ret_Arr[10] := FALSE;
   S703_ELE.Visu_Ret_Arr[11] := FALSE;
   S703_ELE.Visu_Ret_Arr[12] := FALSE;
   S703_ELE.Visu_Ret_Arr[13] := FALSE;
   S703_ELE.Visu_Ret_Arr[14] := FALSE;
   S703_ELE.Visu_Ret_Arr[15] := FALSE;
   S703_ELE.BLK_Move_Ret := 0;
   S703_ELE.Enable := FALSE;
   S703_ELE.Adv_End := FALSE;
   S703_ELE.Ret_End := FALSE;
   S703_AIR_ELE.Enable_Aux := FALSE;
   S703_AIR_ELE.Adv_Amount := 0;
   S703_AIR_ELE.Ret_Amount := 0;
   S703_AIR_ELE.LS_Adv1 := FALSE;
   S703_AIR_ELE.LS_Ret1 := FALSE;
   S703_AIR_ELE.LS_Adv2 := FALSE;
   S703_AIR_ELE.LS_Ret2 := FALSE;
   S703_AIR_ELE.LS_Adv3 := FALSE;
   S703_AIR_ELE.LS_Ret3 := FALSE;
   S703_AIR_ELE.LS_Adv4 := FALSE;
   S703_AIR_ELE.LS_Ret4 := FALSE;
   S703_AIR_ELE.SOL_Adv := FALSE;
   S703_AIR_ELE.SOL_Ret := FALSE;
   S703_AIR_ELE.M_Ready := FALSE;
   S703_AIR_ELE.T_CHK1 := T#0MS;
   S703_AIR_ELE.T_CHK2 := T#0MS;
   S703_AIR_ELE.PB_Lamp_CHK := FALSE;
   S703_AIR_ELE.PB_Error_Rst := FALSE;
   S703_AIR_ELE.M_FLICK := FALSE;
   S703_AIR_ELE.M_Adv_Err := FALSE;
   S703_AIR_ELE.M_Ret_Err := FALSE;
   S703_AIR_ELE.LP_Adv := FALSE;
   S703_AIR_ELE.LP_Ret := FALSE;
   S703_AIR_ELE.Visu_Adv := W#16#0;
   S703_AIR_ELE.Visu_Ret := W#16#0;
   S703_AIR_ELE.Error_T1.IN := FALSE;
   S703_AIR_ELE.Error_T1.PT := T#0MS;
   S703_AIR_ELE.Error_T1.Q := FALSE;
   S703_AIR_ELE.Error_T1.ET := T#0MS;
   S703_AIR_ELE.Error_T1.STATE := B#16#0;
   S703_AIR_ELE.Error_T1.STIME := T#0MS;
   S703_AIR_ELE.Error_T1.ATIME := T#0MS;
   S703_AIR_ELE.Error_T2.IN := FALSE;
   S703_AIR_ELE.Error_T2.PT := T#0MS;
   S703_AIR_ELE.Error_T2.Q := FALSE;
   S703_AIR_ELE.Error_T2.ET := T#0MS;
   S703_AIR_ELE.Error_T2.STATE := B#16#0;
   S703_AIR_ELE.Error_T2.STIME := T#0MS;
   S703_AIR_ELE.Error_T2.ATIME := T#0MS;
   S703_AIR_ELE.CHK_Aux1 := FALSE;
   S703_AIR_ELE.CHK_Aux2 := FALSE;
   S703_AIR_ELE.Error_T1_DN := FALSE;
   S703_AIR_ELE.Error_T2_DN := FALSE;
   S703_AIR_ELE.Adv_Memo := FALSE;
   S703_AIR_ELE.Visu_Adv_Arr[0] := FALSE;
   S703_AIR_ELE.Visu_Adv_Arr[1] := FALSE;
   S703_AIR_ELE.Visu_Adv_Arr[2] := FALSE;
   S703_AIR_ELE.Visu_Adv_Arr[3] := FALSE;
   S703_AIR_ELE.Visu_Adv_Arr[4] := FALSE;
   S703_AIR_ELE.Visu_Adv_Arr[5] := FALSE;
   S703_AIR_ELE.Visu_Adv_Arr[6] := FALSE;
   S703_AIR_ELE.Visu_Adv_Arr[7] := FALSE;
   S703_AIR_ELE.Visu_Adv_Arr[8] := FALSE;
   S703_AIR_ELE.Visu_Adv_Arr[9] := FALSE;
   S703_AIR_ELE.Visu_Adv_Arr[10] := FALSE;
   S703_AIR_ELE.Visu_Adv_Arr[11] := FALSE;
   S703_AIR_ELE.Visu_Adv_Arr[12] := FALSE;
   S703_AIR_ELE.Visu_Adv_Arr[13] := FALSE;
   S703_AIR_ELE.Visu_Adv_Arr[14] := FALSE;
   S703_AIR_ELE.Visu_Adv_Arr[15] := FALSE;
   S703_AIR_ELE.Visu_Ret_Arr[0] := FALSE;
   S703_AIR_ELE.Visu_Ret_Arr[1] := FALSE;
   S703_AIR_ELE.Visu_Ret_Arr[2] := FALSE;
   S703_AIR_ELE.Visu_Ret_Arr[3] := FALSE;
   S703_AIR_ELE.Visu_Ret_Arr[4] := FALSE;
   S703_AIR_ELE.Visu_Ret_Arr[5] := FALSE;
   S703_AIR_ELE.Visu_Ret_Arr[6] := FALSE;
   S703_AIR_ELE.Visu_Ret_Arr[7] := FALSE;
   S703_AIR_ELE.Visu_Ret_Arr[8] := FALSE;
   S703_AIR_ELE.Visu_Ret_Arr[9] := FALSE;
   S703_AIR_ELE.Visu_Ret_Arr[10] := FALSE;
   S703_AIR_ELE.Visu_Ret_Arr[11] := FALSE;
   S703_AIR_ELE.Visu_Ret_Arr[12] := FALSE;
   S703_AIR_ELE.Visu_Ret_Arr[13] := FALSE;
   S703_AIR_ELE.Visu_Ret_Arr[14] := FALSE;
   S703_AIR_ELE.Visu_Ret_Arr[15] := FALSE;
   S703_AIR_ELE.BLK_Move_Ret := 0;
   S703_AIR_ELE.Enable := FALSE;
   S703_AIR_ELE.Adv_End := FALSE;
   S703_AIR_ELE.Ret_End := FALSE;
   S703_ROOF_RACK_A_R.Enable_Aux := FALSE;
   S703_ROOF_RACK_A_R.Adv_Amount := 0;
   S703_ROOF_RACK_A_R.Ret_Amount := 0;
   S703_ROOF_RACK_A_R.LS_Adv1 := FALSE;
   S703_ROOF_RACK_A_R.LS_Ret1 := FALSE;
   S703_ROOF_RACK_A_R.LS_Adv2 := FALSE;
   S703_ROOF_RACK_A_R.LS_Ret2 := FALSE;
   S703_ROOF_RACK_A_R.LS_Adv3 := FALSE;
   S703_ROOF_RACK_A_R.LS_Ret3 := FALSE;
   S703_ROOF_RACK_A_R.LS_Adv4 := FALSE;
   S703_ROOF_RACK_A_R.LS_Ret4 := FALSE;
   S703_ROOF_RACK_A_R.SOL_Adv := FALSE;
   S703_ROOF_RACK_A_R.SOL_Ret := FALSE;
   S703_ROOF_RACK_A_R.M_Ready := FALSE;
   S703_ROOF_RACK_A_R.T_CHK1 := T#0MS;
   S703_ROOF_RACK_A_R.T_CHK2 := T#0MS;
   S703_ROOF_RACK_A_R.PB_Lamp_CHK := FALSE;
   S703_ROOF_RACK_A_R.PB_Error_Rst := FALSE;
   S703_ROOF_RACK_A_R.M_FLICK := FALSE;
   S703_ROOF_RACK_A_R.M_Adv_Err := FALSE;
   S703_ROOF_RACK_A_R.M_Ret_Err := FALSE;
   S703_ROOF_RACK_A_R.LP_Adv := FALSE;
   S703_ROOF_RACK_A_R.LP_Ret := FALSE;
   S703_ROOF_RACK_A_R.Visu_Adv := W#16#0;
   S703_ROOF_RACK_A_R.Visu_Ret := W#16#0;
   S703_ROOF_RACK_A_R.Error_T1.IN := FALSE;
   S703_ROOF_RACK_A_R.Error_T1.PT := T#0MS;
   S703_ROOF_RACK_A_R.Error_T1.Q := FALSE;
   S703_ROOF_RACK_A_R.Error_T1.ET := T#0MS;
   S703_ROOF_RACK_A_R.Error_T1.STATE := B#16#0;
   S703_ROOF_RACK_A_R.Error_T1.STIME := T#0MS;
   S703_ROOF_RACK_A_R.Error_T1.ATIME := T#0MS;
   S703_ROOF_RACK_A_R.Error_T2.IN := FALSE;
   S703_ROOF_RACK_A_R.Error_T2.PT := T#0MS;
   S703_ROOF_RACK_A_R.Error_T2.Q := FALSE;
   S703_ROOF_RACK_A_R.Error_T2.ET := T#0MS;
   S703_ROOF_RACK_A_R.Error_T2.STATE := B#16#0;
   S703_ROOF_RACK_A_R.Error_T2.STIME := T#0MS;
   S703_ROOF_RACK_A_R.Error_T2.ATIME := T#0MS;
   S703_ROOF_RACK_A_R.CHK_Aux1 := FALSE;
   S703_ROOF_RACK_A_R.CHK_Aux2 := FALSE;
   S703_ROOF_RACK_A_R.Error_T1_DN := FALSE;
   S703_ROOF_RACK_A_R.Error_T2_DN := FALSE;
   S703_ROOF_RACK_A_R.Adv_Memo := FALSE;
   S703_ROOF_RACK_A_R.Visu_Adv_Arr[0] := FALSE;
   S703_ROOF_RACK_A_R.Visu_Adv_Arr[1] := FALSE;
   S703_ROOF_RACK_A_R.Visu_Adv_Arr[2] := FALSE;
   S703_ROOF_RACK_A_R.Visu_Adv_Arr[3] := FALSE;
   S703_ROOF_RACK_A_R.Visu_Adv_Arr[4] := FALSE;
   S703_ROOF_RACK_A_R.Visu_Adv_Arr[5] := FALSE;
   S703_ROOF_RACK_A_R.Visu_Adv_Arr[6] := FALSE;
   S703_ROOF_RACK_A_R.Visu_Adv_Arr[7] := FALSE;
   S703_ROOF_RACK_A_R.Visu_Adv_Arr[8] := FALSE;
   S703_ROOF_RACK_A_R.Visu_Adv_Arr[9] := FALSE;
   S703_ROOF_RACK_A_R.Visu_Adv_Arr[10] := FALSE;
   S703_ROOF_RACK_A_R.Visu_Adv_Arr[11] := FALSE;
   S703_ROOF_RACK_A_R.Visu_Adv_Arr[12] := FALSE;
   S703_ROOF_RACK_A_R.Visu_Adv_Arr[13] := FALSE;
   S703_ROOF_RACK_A_R.Visu_Adv_Arr[14] := FALSE;
   S703_ROOF_RACK_A_R.Visu_Adv_Arr[15] := FALSE;
   S703_ROOF_RACK_A_R.Visu_Ret_Arr[0] := FALSE;
   S703_ROOF_RACK_A_R.Visu_Ret_Arr[1] := FALSE;
   S703_ROOF_RACK_A_R.Visu_Ret_Arr[2] := FALSE;
   S703_ROOF_RACK_A_R.Visu_Ret_Arr[3] := FALSE;
   S703_ROOF_RACK_A_R.Visu_Ret_Arr[4] := FALSE;
   S703_ROOF_RACK_A_R.Visu_Ret_Arr[5] := FALSE;
   S703_ROOF_RACK_A_R.Visu_Ret_Arr[6] := FALSE;
   S703_ROOF_RACK_A_R.Visu_Ret_Arr[7] := FALSE;
   S703_ROOF_RACK_A_R.Visu_Ret_Arr[8] := FALSE;
   S703_ROOF_RACK_A_R.Visu_Ret_Arr[9] := FALSE;
   S703_ROOF_RACK_A_R.Visu_Ret_Arr[10] := FALSE;
   S703_ROOF_RACK_A_R.Visu_Ret_Arr[11] := FALSE;
   S703_ROOF_RACK_A_R.Visu_Ret_Arr[12] := FALSE;
   S703_ROOF_RACK_A_R.Visu_Ret_Arr[13] := FALSE;
   S703_ROOF_RACK_A_R.Visu_Ret_Arr[14] := FALSE;
   S703_ROOF_RACK_A_R.Visu_Ret_Arr[15] := FALSE;
   S703_ROOF_RACK_A_R.BLK_Move_Ret := 0;
   S703_ROOF_RACK_A_R.Enable := FALSE;
   S703_ROOF_RACK_A_R.Adv_End := FALSE;
   S703_ROOF_RACK_A_R.Ret_End := FALSE;
   S703_ROOF_RACK_CLAMP.Enable_Aux := FALSE;
   S703_ROOF_RACK_CLAMP.Adv_Amount := 0;
   S703_ROOF_RACK_CLAMP.Ret_Amount := 0;
   S703_ROOF_RACK_CLAMP.LS_Adv1 := FALSE;
   S703_ROOF_RACK_CLAMP.LS_Ret1 := FALSE;
   S703_ROOF_RACK_CLAMP.LS_Adv2 := FALSE;
   S703_ROOF_RACK_CLAMP.LS_Ret2 := FALSE;
   S703_ROOF_RACK_CLAMP.LS_Adv3 := FALSE;
   S703_ROOF_RACK_CLAMP.LS_Ret3 := FALSE;
   S703_ROOF_RACK_CLAMP.LS_Adv4 := FALSE;
   S703_ROOF_RACK_CLAMP.LS_Ret4 := FALSE;
   S703_ROOF_RACK_CLAMP.SOL_Adv := FALSE;
   S703_ROOF_RACK_CLAMP.SOL_Ret := FALSE;
   S703_ROOF_RACK_CLAMP.M_Ready := FALSE;
   S703_ROOF_RACK_CLAMP.T_CHK1 := T#0MS;
   S703_ROOF_RACK_CLAMP.T_CHK2 := T#0MS;
   S703_ROOF_RACK_CLAMP.PB_Lamp_CHK := FALSE;
   S703_ROOF_RACK_CLAMP.PB_Error_Rst := FALSE;
   S703_ROOF_RACK_CLAMP.M_FLICK := FALSE;
   S703_ROOF_RACK_CLAMP.M_Adv_Err := FALSE;
   S703_ROOF_RACK_CLAMP.M_Ret_Err := FALSE;
   S703_ROOF_RACK_CLAMP.LP_Adv := FALSE;
   S703_ROOF_RACK_CLAMP.LP_Ret := FALSE;
   S703_ROOF_RACK_CLAMP.Visu_Adv := W#16#0;
   S703_ROOF_RACK_CLAMP.Visu_Ret := W#16#0;
   S703_ROOF_RACK_CLAMP.Error_T1.IN := FALSE;
   S703_ROOF_RACK_CLAMP.Error_T1.PT := T#0MS;
   S703_ROOF_RACK_CLAMP.Error_T1.Q := FALSE;
   S703_ROOF_RACK_CLAMP.Error_T1.ET := T#0MS;
   S703_ROOF_RACK_CLAMP.Error_T1.STATE := B#16#0;
   S703_ROOF_RACK_CLAMP.Error_T1.STIME := T#0MS;
   S703_ROOF_RACK_CLAMP.Error_T1.ATIME := T#0MS;
   S703_ROOF_RACK_CLAMP.Error_T2.IN := FALSE;
   S703_ROOF_RACK_CLAMP.Error_T2.PT := T#0MS;
   S703_ROOF_RACK_CLAMP.Error_T2.Q := FALSE;
   S703_ROOF_RACK_CLAMP.Error_T2.ET := T#0MS;
   S703_ROOF_RACK_CLAMP.Error_T2.STATE := B#16#0;
   S703_ROOF_RACK_CLAMP.Error_T2.STIME := T#0MS;
   S703_ROOF_RACK_CLAMP.Error_T2.ATIME := T#0MS;
   S703_ROOF_RACK_CLAMP.CHK_Aux1 := FALSE;
   S703_ROOF_RACK_CLAMP.CHK_Aux2 := FALSE;
   S703_ROOF_RACK_CLAMP.Error_T1_DN := FALSE;
   S703_ROOF_RACK_CLAMP.Error_T2_DN := FALSE;
   S703_ROOF_RACK_CLAMP.Adv_Memo := FALSE;
   S703_ROOF_RACK_CLAMP.Visu_Adv_Arr[0] := FALSE;
   S703_ROOF_RACK_CLAMP.Visu_Adv_Arr[1] := FALSE;
   S703_ROOF_RACK_CLAMP.Visu_Adv_Arr[2] := FALSE;
   S703_ROOF_RACK_CLAMP.Visu_Adv_Arr[3] := FALSE;
   S703_ROOF_RACK_CLAMP.Visu_Adv_Arr[4] := FALSE;
   S703_ROOF_RACK_CLAMP.Visu_Adv_Arr[5] := FALSE;
   S703_ROOF_RACK_CLAMP.Visu_Adv_Arr[6] := FALSE;
   S703_ROOF_RACK_CLAMP.Visu_Adv_Arr[7] := FALSE;
   S703_ROOF_RACK_CLAMP.Visu_Adv_Arr[8] := FALSE;
   S703_ROOF_RACK_CLAMP.Visu_Adv_Arr[9] := FALSE;
   S703_ROOF_RACK_CLAMP.Visu_Adv_Arr[10] := FALSE;
   S703_ROOF_RACK_CLAMP.Visu_Adv_Arr[11] := FALSE;
   S703_ROOF_RACK_CLAMP.Visu_Adv_Arr[12] := FALSE;
   S703_ROOF_RACK_CLAMP.Visu_Adv_Arr[13] := FALSE;
   S703_ROOF_RACK_CLAMP.Visu_Adv_Arr[14] := FALSE;
   S703_ROOF_RACK_CLAMP.Visu_Adv_Arr[15] := FALSE;
   S703_ROOF_RACK_CLAMP.Visu_Ret_Arr[0] := FALSE;
   S703_ROOF_RACK_CLAMP.Visu_Ret_Arr[1] := FALSE;
   S703_ROOF_RACK_CLAMP.Visu_Ret_Arr[2] := FALSE;
   S703_ROOF_RACK_CLAMP.Visu_Ret_Arr[3] := FALSE;
   S703_ROOF_RACK_CLAMP.Visu_Ret_Arr[4] := FALSE;
   S703_ROOF_RACK_CLAMP.Visu_Ret_Arr[5] := FALSE;
   S703_ROOF_RACK_CLAMP.Visu_Ret_Arr[6] := FALSE;
   S703_ROOF_RACK_CLAMP.Visu_Ret_Arr[7] := FALSE;
   S703_ROOF_RACK_CLAMP.Visu_Ret_Arr[8] := FALSE;
   S703_ROOF_RACK_CLAMP.Visu_Ret_Arr[9] := FALSE;
   S703_ROOF_RACK_CLAMP.Visu_Ret_Arr[10] := FALSE;
   S703_ROOF_RACK_CLAMP.Visu_Ret_Arr[11] := FALSE;
   S703_ROOF_RACK_CLAMP.Visu_Ret_Arr[12] := FALSE;
   S703_ROOF_RACK_CLAMP.Visu_Ret_Arr[13] := FALSE;
   S703_ROOF_RACK_CLAMP.Visu_Ret_Arr[14] := FALSE;
   S703_ROOF_RACK_CLAMP.Visu_Ret_Arr[15] := FALSE;
   S703_ROOF_RACK_CLAMP.BLK_Move_Ret := 0;
   S703_ROOF_RACK_CLAMP.Enable := FALSE;
   S703_ROOF_RACK_CLAMP.Adv_End := FALSE;
   S703_ROOF_RACK_CLAMP.Ret_End := FALSE;
   S703_ROOF_RACK_GUN1_A_R.Enable_Aux := FALSE;
   S703_ROOF_RACK_GUN1_A_R.Adv_Amount := 0;
   S703_ROOF_RACK_GUN1_A_R.Ret_Amount := 0;
   S703_ROOF_RACK_GUN1_A_R.LS_Adv1 := FALSE;
   S703_ROOF_RACK_GUN1_A_R.LS_Ret1 := FALSE;
   S703_ROOF_RACK_GUN1_A_R.LS_Adv2 := FALSE;
   S703_ROOF_RACK_GUN1_A_R.LS_Ret2 := FALSE;
   S703_ROOF_RACK_GUN1_A_R.LS_Adv3 := FALSE;
   S703_ROOF_RACK_GUN1_A_R.LS_Ret3 := FALSE;
   S703_ROOF_RACK_GUN1_A_R.LS_Adv4 := FALSE;
   S703_ROOF_RACK_GUN1_A_R.LS_Ret4 := FALSE;
   S703_ROOF_RACK_GUN1_A_R.SOL_Adv := FALSE;
   S703_ROOF_RACK_GUN1_A_R.SOL_Ret := FALSE;
   S703_ROOF_RACK_GUN1_A_R.M_Ready := FALSE;
   S703_ROOF_RACK_GUN1_A_R.T_CHK1 := T#0MS;
   S703_ROOF_RACK_GUN1_A_R.T_CHK2 := T#0MS;
   S703_ROOF_RACK_GUN1_A_R.PB_Lamp_CHK := FALSE;
   S703_ROOF_RACK_GUN1_A_R.PB_Error_Rst := FALSE;
   S703_ROOF_RACK_GUN1_A_R.M_FLICK := FALSE;
   S703_ROOF_RACK_GUN1_A_R.M_Adv_Err := FALSE;
   S703_ROOF_RACK_GUN1_A_R.M_Ret_Err := FALSE;
   S703_ROOF_RACK_GUN1_A_R.LP_Adv := FALSE;
   S703_ROOF_RACK_GUN1_A_R.LP_Ret := FALSE;
   S703_ROOF_RACK_GUN1_A_R.Visu_Adv := W#16#0;
   S703_ROOF_RACK_GUN1_A_R.Visu_Ret := W#16#0;
   S703_ROOF_RACK_GUN1_A_R.Error_T1.IN := FALSE;
   S703_ROOF_RACK_GUN1_A_R.Error_T1.PT := T#0MS;
   S703_ROOF_RACK_GUN1_A_R.Error_T1.Q := FALSE;
   S703_ROOF_RACK_GUN1_A_R.Error_T1.ET := T#0MS;
   S703_ROOF_RACK_GUN1_A_R.Error_T1.STATE := B#16#0;
   S703_ROOF_RACK_GUN1_A_R.Error_T1.STIME := T#0MS;
   S703_ROOF_RACK_GUN1_A_R.Error_T1.ATIME := T#0MS;
   S703_ROOF_RACK_GUN1_A_R.Error_T2.IN := FALSE;
   S703_ROOF_RACK_GUN1_A_R.Error_T2.PT := T#0MS;
   S703_ROOF_RACK_GUN1_A_R.Error_T2.Q := FALSE;
   S703_ROOF_RACK_GUN1_A_R.Error_T2.ET := T#0MS;
   S703_ROOF_RACK_GUN1_A_R.Error_T2.STATE := B#16#0;
   S703_ROOF_RACK_GUN1_A_R.Error_T2.STIME := T#0MS;
   S703_ROOF_RACK_GUN1_A_R.Error_T2.ATIME := T#0MS;
   S703_ROOF_RACK_GUN1_A_R.CHK_Aux1 := FALSE;
   S703_ROOF_RACK_GUN1_A_R.CHK_Aux2 := FALSE;
   S703_ROOF_RACK_GUN1_A_R.Error_T1_DN := FALSE;
   S703_ROOF_RACK_GUN1_A_R.Error_T2_DN := FALSE;
   S703_ROOF_RACK_GUN1_A_R.Adv_Memo := FALSE;
   S703_ROOF_RACK_GUN1_A_R.Visu_Adv_Arr[0] := FALSE;
   S703_ROOF_RACK_GUN1_A_R.Visu_Adv_Arr[1] := FALSE;
   S703_ROOF_RACK_GUN1_A_R.Visu_Adv_Arr[2] := FALSE;
   S703_ROOF_RACK_GUN1_A_R.Visu_Adv_Arr[3] := FALSE;
   S703_ROOF_RACK_GUN1_A_R.Visu_Adv_Arr[4] := FALSE;
   S703_ROOF_RACK_GUN1_A_R.Visu_Adv_Arr[5] := FALSE;
   S703_ROOF_RACK_GUN1_A_R.Visu_Adv_Arr[6] := FALSE;
   S703_ROOF_RACK_GUN1_A_R.Visu_Adv_Arr[7] := FALSE;
   S703_ROOF_RACK_GUN1_A_R.Visu_Adv_Arr[8] := FALSE;
   S703_ROOF_RACK_GUN1_A_R.Visu_Adv_Arr[9] := FALSE;
   S703_ROOF_RACK_GUN1_A_R.Visu_Adv_Arr[10] := FALSE;
   S703_ROOF_RACK_GUN1_A_R.Visu_Adv_Arr[11] := FALSE;
   S703_ROOF_RACK_GUN1_A_R.Visu_Adv_Arr[12] := FALSE;
   S703_ROOF_RACK_GUN1_A_R.Visu_Adv_Arr[13] := FALSE;
   S703_ROOF_RACK_GUN1_A_R.Visu_Adv_Arr[14] := FALSE;
   S703_ROOF_RACK_GUN1_A_R.Visu_Adv_Arr[15] := FALSE;
   S703_ROOF_RACK_GUN1_A_R.Visu_Ret_Arr[0] := FALSE;
   S703_ROOF_RACK_GUN1_A_R.Visu_Ret_Arr[1] := FALSE;
   S703_ROOF_RACK_GUN1_A_R.Visu_Ret_Arr[2] := FALSE;
   S703_ROOF_RACK_GUN1_A_R.Visu_Ret_Arr[3] := FALSE;
   S703_ROOF_RACK_GUN1_A_R.Visu_Ret_Arr[4] := FALSE;
   S703_ROOF_RACK_GUN1_A_R.Visu_Ret_Arr[5] := FALSE;
   S703_ROOF_RACK_GUN1_A_R.Visu_Ret_Arr[6] := FALSE;
   S703_ROOF_RACK_GUN1_A_R.Visu_Ret_Arr[7] := FALSE;
   S703_ROOF_RACK_GUN1_A_R.Visu_Ret_Arr[8] := FALSE;
   S703_ROOF_RACK_GUN1_A_R.Visu_Ret_Arr[9] := FALSE;
   S703_ROOF_RACK_GUN1_A_R.Visu_Ret_Arr[10] := FALSE;
   S703_ROOF_RACK_GUN1_A_R.Visu_Ret_Arr[11] := FALSE;
   S703_ROOF_RACK_GUN1_A_R.Visu_Ret_Arr[12] := FALSE;
   S703_ROOF_RACK_GUN1_A_R.Visu_Ret_Arr[13] := FALSE;
   S703_ROOF_RACK_GUN1_A_R.Visu_Ret_Arr[14] := FALSE;
   S703_ROOF_RACK_GUN1_A_R.Visu_Ret_Arr[15] := FALSE;
   S703_ROOF_RACK_GUN1_A_R.BLK_Move_Ret := 0;
   S703_ROOF_RACK_GUN1_A_R.Enable := FALSE;
   S703_ROOF_RACK_GUN1_A_R.Adv_End := FALSE;
   S703_ROOF_RACK_GUN1_A_R.Ret_End := FALSE;
   S703_ROOF_RACK_GUN2_A_R.Enable_Aux := FALSE;
   S703_ROOF_RACK_GUN2_A_R.Adv_Amount := 0;
   S703_ROOF_RACK_GUN2_A_R.Ret_Amount := 0;
   S703_ROOF_RACK_GUN2_A_R.LS_Adv1 := FALSE;
   S703_ROOF_RACK_GUN2_A_R.LS_Ret1 := FALSE;
   S703_ROOF_RACK_GUN2_A_R.LS_Adv2 := FALSE;
   S703_ROOF_RACK_GUN2_A_R.LS_Ret2 := FALSE;
   S703_ROOF_RACK_GUN2_A_R.LS_Adv3 := FALSE;
   S703_ROOF_RACK_GUN2_A_R.LS_Ret3 := FALSE;
   S703_ROOF_RACK_GUN2_A_R.LS_Adv4 := FALSE;
   S703_ROOF_RACK_GUN2_A_R.LS_Ret4 := FALSE;
   S703_ROOF_RACK_GUN2_A_R.SOL_Adv := FALSE;
   S703_ROOF_RACK_GUN2_A_R.SOL_Ret := FALSE;
   S703_ROOF_RACK_GUN2_A_R.M_Ready := FALSE;
   S703_ROOF_RACK_GUN2_A_R.T_CHK1 := T#0MS;
   S703_ROOF_RACK_GUN2_A_R.T_CHK2 := T#0MS;
   S703_ROOF_RACK_GUN2_A_R.PB_Lamp_CHK := FALSE;
   S703_ROOF_RACK_GUN2_A_R.PB_Error_Rst := FALSE;
   S703_ROOF_RACK_GUN2_A_R.M_FLICK := FALSE;
   S703_ROOF_RACK_GUN2_A_R.M_Adv_Err := FALSE;
   S703_ROOF_RACK_GUN2_A_R.M_Ret_Err := FALSE;
   S703_ROOF_RACK_GUN2_A_R.LP_Adv := FALSE;
   S703_ROOF_RACK_GUN2_A_R.LP_Ret := FALSE;
   S703_ROOF_RACK_GUN2_A_R.Visu_Adv := W#16#0;
   S703_ROOF_RACK_GUN2_A_R.Visu_Ret := W#16#0;
   S703_ROOF_RACK_GUN2_A_R.Error_T1.IN := FALSE;
   S703_ROOF_RACK_GUN2_A_R.Error_T1.PT := T#0MS;
   S703_ROOF_RACK_GUN2_A_R.Error_T1.Q := FALSE;
   S703_ROOF_RACK_GUN2_A_R.Error_T1.ET := T#0MS;
   S703_ROOF_RACK_GUN2_A_R.Error_T1.STATE := B#16#0;
   S703_ROOF_RACK_GUN2_A_R.Error_T1.STIME := T#0MS;
   S703_ROOF_RACK_GUN2_A_R.Error_T1.ATIME := T#0MS;
   S703_ROOF_RACK_GUN2_A_R.Error_T2.IN := FALSE;
   S703_ROOF_RACK_GUN2_A_R.Error_T2.PT := T#0MS;
   S703_ROOF_RACK_GUN2_A_R.Error_T2.Q := FALSE;
   S703_ROOF_RACK_GUN2_A_R.Error_T2.ET := T#0MS;
   S703_ROOF_RACK_GUN2_A_R.Error_T2.STATE := B#16#0;
   S703_ROOF_RACK_GUN2_A_R.Error_T2.STIME := T#0MS;
   S703_ROOF_RACK_GUN2_A_R.Error_T2.ATIME := T#0MS;
   S703_ROOF_RACK_GUN2_A_R.CHK_Aux1 := FALSE;
   S703_ROOF_RACK_GUN2_A_R.CHK_Aux2 := FALSE;
   S703_ROOF_RACK_GUN2_A_R.Error_T1_DN := FALSE;
   S703_ROOF_RACK_GUN2_A_R.Error_T2_DN := FALSE;
   S703_ROOF_RACK_GUN2_A_R.Adv_Memo := FALSE;
   S703_ROOF_RACK_GUN2_A_R.Visu_Adv_Arr[0] := FALSE;
   S703_ROOF_RACK_GUN2_A_R.Visu_Adv_Arr[1] := FALSE;
   S703_ROOF_RACK_GUN2_A_R.Visu_Adv_Arr[2] := FALSE;
   S703_ROOF_RACK_GUN2_A_R.Visu_Adv_Arr[3] := FALSE;
   S703_ROOF_RACK_GUN2_A_R.Visu_Adv_Arr[4] := FALSE;
   S703_ROOF_RACK_GUN2_A_R.Visu_Adv_Arr[5] := FALSE;
   S703_ROOF_RACK_GUN2_A_R.Visu_Adv_Arr[6] := FALSE;
   S703_ROOF_RACK_GUN2_A_R.Visu_Adv_Arr[7] := FALSE;
   S703_ROOF_RACK_GUN2_A_R.Visu_Adv_Arr[8] := FALSE;
   S703_ROOF_RACK_GUN2_A_R.Visu_Adv_Arr[9] := FALSE;
   S703_ROOF_RACK_GUN2_A_R.Visu_Adv_Arr[10] := FALSE;
   S703_ROOF_RACK_GUN2_A_R.Visu_Adv_Arr[11] := FALSE;
   S703_ROOF_RACK_GUN2_A_R.Visu_Adv_Arr[12] := FALSE;
   S703_ROOF_RACK_GUN2_A_R.Visu_Adv_Arr[13] := FALSE;
   S703_ROOF_RACK_GUN2_A_R.Visu_Adv_Arr[14] := FALSE;
   S703_ROOF_RACK_GUN2_A_R.Visu_Adv_Arr[15] := FALSE;
   S703_ROOF_RACK_GUN2_A_R.Visu_Ret_Arr[0] := FALSE;
   S703_ROOF_RACK_GUN2_A_R.Visu_Ret_Arr[1] := FALSE;
   S703_ROOF_RACK_GUN2_A_R.Visu_Ret_Arr[2] := FALSE;
   S703_ROOF_RACK_GUN2_A_R.Visu_Ret_Arr[3] := FALSE;
   S703_ROOF_RACK_GUN2_A_R.Visu_Ret_Arr[4] := FALSE;
   S703_ROOF_RACK_GUN2_A_R.Visu_Ret_Arr[5] := FALSE;
   S703_ROOF_RACK_GUN2_A_R.Visu_Ret_Arr[6] := FALSE;
   S703_ROOF_RACK_GUN2_A_R.Visu_Ret_Arr[7] := FALSE;
   S703_ROOF_RACK_GUN2_A_R.Visu_Ret_Arr[8] := FALSE;
   S703_ROOF_RACK_GUN2_A_R.Visu_Ret_Arr[9] := FALSE;
   S703_ROOF_RACK_GUN2_A_R.Visu_Ret_Arr[10] := FALSE;
   S703_ROOF_RACK_GUN2_A_R.Visu_Ret_Arr[11] := FALSE;
   S703_ROOF_RACK_GUN2_A_R.Visu_Ret_Arr[12] := FALSE;
   S703_ROOF_RACK_GUN2_A_R.Visu_Ret_Arr[13] := FALSE;
   S703_ROOF_RACK_GUN2_A_R.Visu_Ret_Arr[14] := FALSE;
   S703_ROOF_RACK_GUN2_A_R.Visu_Ret_Arr[15] := FALSE;
   S703_ROOF_RACK_GUN2_A_R.BLK_Move_Ret := 0;
   S703_ROOF_RACK_GUN2_A_R.Enable := FALSE;
   S703_ROOF_RACK_GUN2_A_R.Adv_End := FALSE;
   S703_ROOF_RACK_GUN2_A_R.Ret_End := FALSE;
END_DATA_BLOCK

FUNCTION FC 131 : VOID
TITLE =
VERSION : 0.1

BEGIN
NETWORK
TITLE =
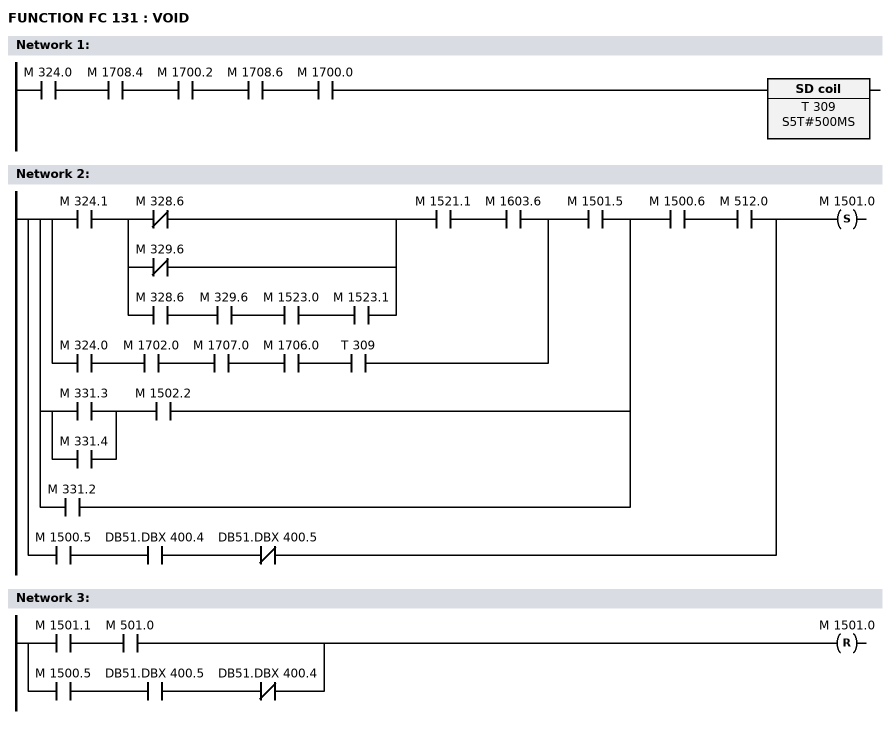

      A     M    324.0;
      A     M   1708.4;
      A     M   1700.2;
      A     M   1708.6;
      A     M   1700.0;
      L     S5T#500MS;
      SD    T    309;
NETWORK
TITLE =

      A(    ;
      A(    ;
      A     M    324.1;
      A(    ;
      ON    M    328.6;
      ON    M    329.6;
      O     ;
      A     M    328.6;
      A     M    329.6;
      A     M   1523.0;
      A     M   1523.1;
      )     ;
      A     M   1521.1;
      A     M   1603.6;
      O     ;
      A     M    324.0;
      A     M   1702.0;
      A     M   1707.0;
      A     M   1706.0;
      A     T    309;
      )     ;
      A     M   1501.5;
      O     ;
      A(    ;
      O     M    331.3;
      O     M    331.4;
      )     ;
      A     M   1502.2;
      O     M    331.2;
      )     ;
      A     M   1500.6;
      A     M    512.0;
      O     ;
      A     M   1500.5;
      A     DB51.DBX  400.4;
      AN    DB51.DBX  400.5;
      S     M   1501.0;
NETWORK
TITLE =

      A     M   1501.1;
      A     M    501.0;
      O     ;
      A     M   1500.5;
      A     DB51.DBX  400.5;
      AN    DB51.DBX  400.4;
      R     M   1501.0;
END_FUNCTION

FUNCTION_BLOCK FB 132
TITLE =
VERSION : 0.1

BEGIN
NETWORK
TITLE =
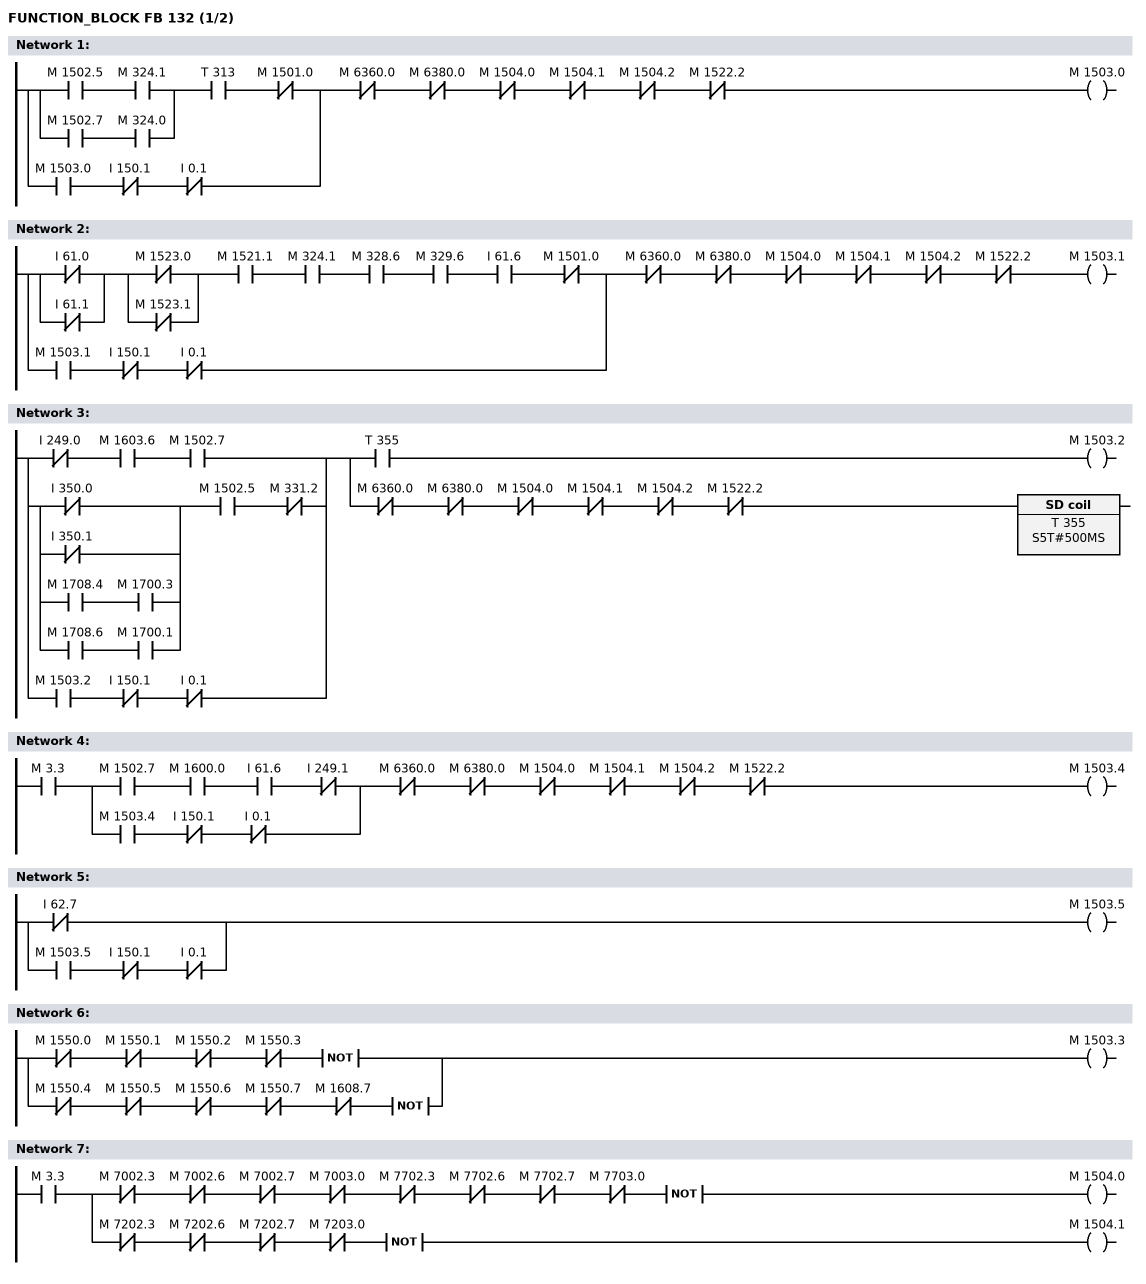

      A(    ;
      A(    ;
      A     M   1502.5;
      A     M    324.1;
      O     ;
      A     M   1502.7;
      A     M    324.0;
      )     ;
      A     T    313;
      AN    M   1501.0;
      O     ;
      A     M   1503.0;
      AN    I    150.1;
      AN    I      0.1;
      )     ;
      AN    M   6360.0;
      AN    M   6380.0;
      AN    M   1504.0;
      AN    M   1504.1;
      AN    M   1504.2;
      AN    M   1522.2;
      =     M   1503.0;
NETWORK
TITLE =

      A(    ;
      A(    ;
      ON    I     61.0;
      ON    I     61.1;
      )     ;
      A(    ;
      ON    M   1523.0;
      ON    M   1523.1;
      )     ;
      A     M   1521.1;
      A     M    324.1;
      A     M    328.6;
      A     M    329.6;
      A     I     61.6;
      AN    M   1501.0;
      O     ;
      A     M   1503.1;
      AN    I    150.1;
      AN    I      0.1;
      )     ;
      AN    M   6360.0;
      AN    M   6380.0;
      AN    M   1504.0;
      AN    M   1504.1;
      AN    M   1504.2;
      AN    M   1522.2;
      =     M   1503.1;
NETWORK
TITLE =

      AN    I    249.0;
      A     M   1603.6;
      A     M   1502.7;
      O     ;
      A(    ;
      ON    I    350.0;
      ON    I    350.1;
      O     ;
      A     M   1708.4;
      A     M   1700.3;
      O     ;
      A     M   1708.6;
      A     M   1700.1;
      )     ;
      A     M   1502.5;
      AN    M    331.2;
      O     ;
      A     M   1503.2;
      AN    I    150.1;
      AN    I      0.1;
      =     L      0.0;
      A     L      0.0;
      A     T    355;
      =     M   1503.2;
      A     L      0.0;
      AN    M   6360.0;
      AN    M   6380.0;
      AN    M   1504.0;
      AN    M   1504.1;
      AN    M   1504.2;
      AN    M   1522.2;
      L     S5T#500MS;
      SD    T    355;
NETWORK
TITLE =

      A     M      3.3;
      A(    ;
      A     M   1502.7;
      A     M   1600.0;
      A     I     61.6;
      AN    I    249.1;
      O     ;
      A     M   1503.4;
      AN    I    150.1;
      AN    I      0.1;
      )     ;
      AN    M   6360.0;
      AN    M   6380.0;
      AN    M   1504.0;
      AN    M   1504.1;
      AN    M   1504.2;
      AN    M   1522.2;
      =     M   1503.4;
NETWORK
TITLE =

      ON    I     62.7;
      O     ;
      A     M   1503.5;
      AN    I    150.1;
      AN    I      0.1;
      =     M   1503.5;
NETWORK
TITLE =

      AN    M   1550.0;
      AN    M   1550.1;
      AN    M   1550.2;
      AN    M   1550.3;
      NOT   ;
      O(    ;
      AN    M   1550.4;
      AN    M   1550.5;
      AN    M   1550.6;
      AN    M   1550.7;
      AN    M   1608.7;
      NOT   ;
      )     ;
      =     M   1503.3;
NETWORK
TITLE =

      A     M      3.3;
      =     L      0.0;
      A     L      0.0;
      AN    M   7002.3;
      AN    M   7002.6;
      AN    M   7002.7;
      AN    M   7003.0;
      AN    M   7702.3;
      AN    M   7702.6;
      AN    M   7702.7;
      AN    M   7703.0;
      NOT   ;
      =     M   1504.0;
      A     L      0.0;
      AN    M   7202.3;
      AN    M   7202.6;
      AN    M   7202.7;
      AN    M   7203.0;
      NOT   ;
      =     M   1504.1;
NETWORK
TITLE =
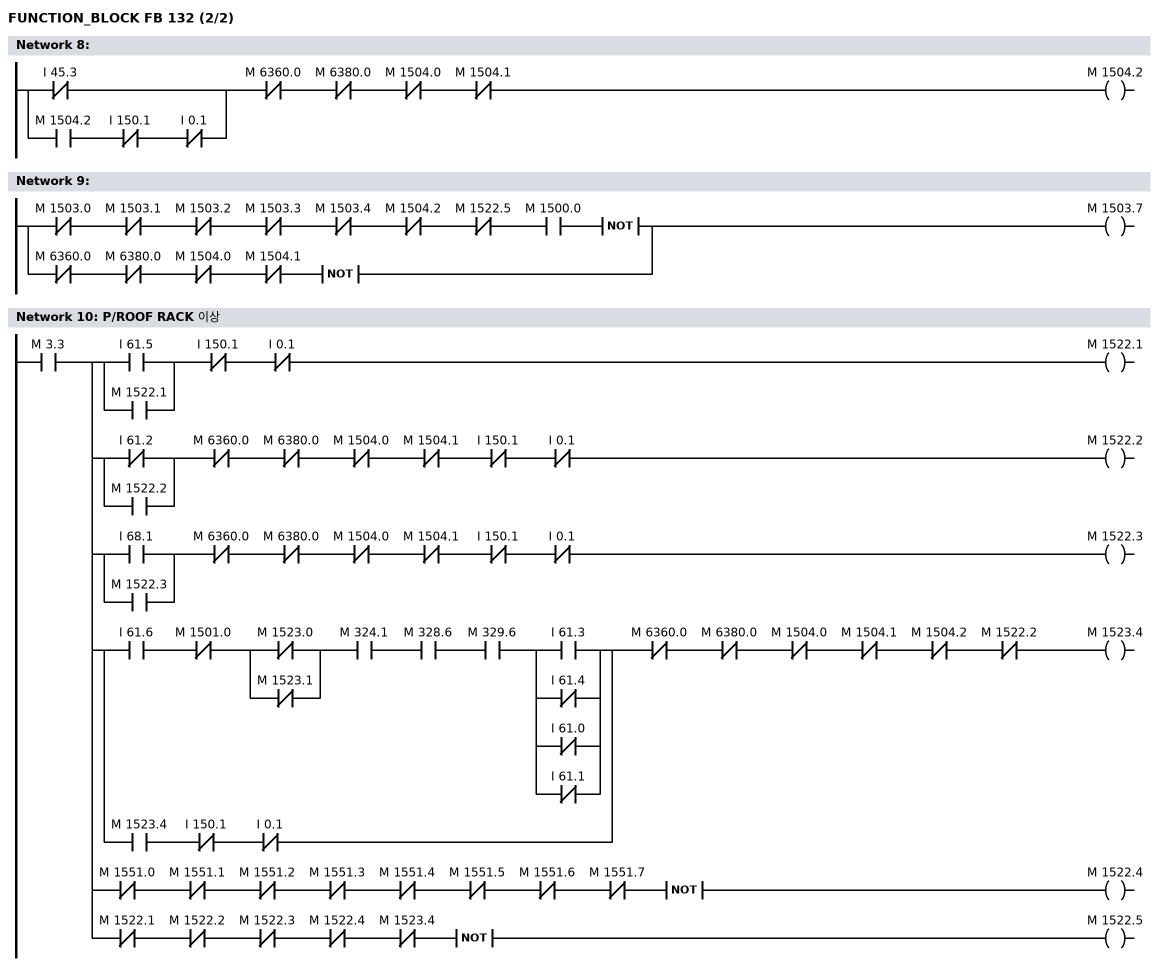

      A(    ;
      ON    I     45.3;
      O     ;
      A     M   1504.2;
      AN    I    150.1;
      AN    I      0.1;
      )     ;
      AN    M   6360.0;
      AN    M   6380.0;
      AN    M   1504.0;
      AN    M   1504.1;
      =     M   1504.2;
NETWORK
TITLE =

      AN    M   1503.0;
      AN    M   1503.1;
      AN    M   1503.2;
      AN    M   1503.3;
      AN    M   1503.4;
      AN    M   1504.2;
      AN    M   1522.5;
      A     M   1500.0;
      NOT   ;
      O(    ;
      AN    M   6360.0;
      AN    M   6380.0;
      AN    M   1504.0;
      AN    M   1504.1;
      NOT   ;
      )     ;
      =     M   1503.7;
NETWORK
TITLE =P/ROOF RACK 이상

      A     M      3.3;
      =     L      0.0;
      A     L      0.0;
      A(    ;
      O     I     61.5;
      O     M   1522.1;
      )     ;
      AN    I    150.1;
      AN    I      0.1;
      =     M   1522.1;
      A     L      0.0;
      A(    ;
      ON    I     61.2;
      O     M   1522.2;
      )     ;
      AN    M   6360.0;
      AN    M   6380.0;
      AN    M   1504.0;
      AN    M   1504.1;
      AN    I    150.1;
      AN    I      0.1;
      =     M   1522.2;
      A     L      0.0;
      A(    ;
      O     I     68.1;
      O     M   1522.3;
      )     ;
      AN    M   6360.0;
      AN    M   6380.0;
      AN    M   1504.0;
      AN    M   1504.1;
      AN    I    150.1;
      AN    I      0.1;
      =     M   1522.3;
      A     L      0.0;
      A(    ;
      A     I     61.6;
      AN    M   1501.0;
      A(    ;
      ON    M   1523.0;
      ON    M   1523.1;
      )     ;
      A     M    324.1;
      A     M    328.6;
      A     M    329.6;
      A(    ;
      O     I     61.3;
      ON    I     61.4;
      ON    I     61.0;
      ON    I     61.1;
      )     ;
      O     ;
      A     M   1523.4;
      AN    I    150.1;
      AN    I      0.1;
      )     ;
      AN    M   6360.0;
      AN    M   6380.0;
      AN    M   1504.0;
      AN    M   1504.1;
      AN    M   1504.2;
      AN    M   1522.2;
      =     M   1523.4;
      A     L      0.0;
      AN    M   1551.0;
      AN    M   1551.1;
      AN    M   1551.2;
      AN    M   1551.3;
      AN    M   1551.4;
      AN    M   1551.5;
      AN    M   1551.6;
      AN    M   1551.7;
      NOT   ;
      =     M   1522.4;
      A     L      0.0;
      AN    M   1522.1;
      AN    M   1522.2;
      AN    M   1522.3;
      AN    M   1522.4;
      AN    M   1523.4;
      NOT   ;
      =     M   1522.5;
END_FUNCTION_BLOCK

DATA_BLOCK DB 132
TITLE =
VERSION : 0.0

 FB 132
BEGIN
END_DATA_BLOCK

FUNCTION FC 132 : VOID
TITLE =
VERSION : 0.1

BEGIN
NETWORK
TITLE =
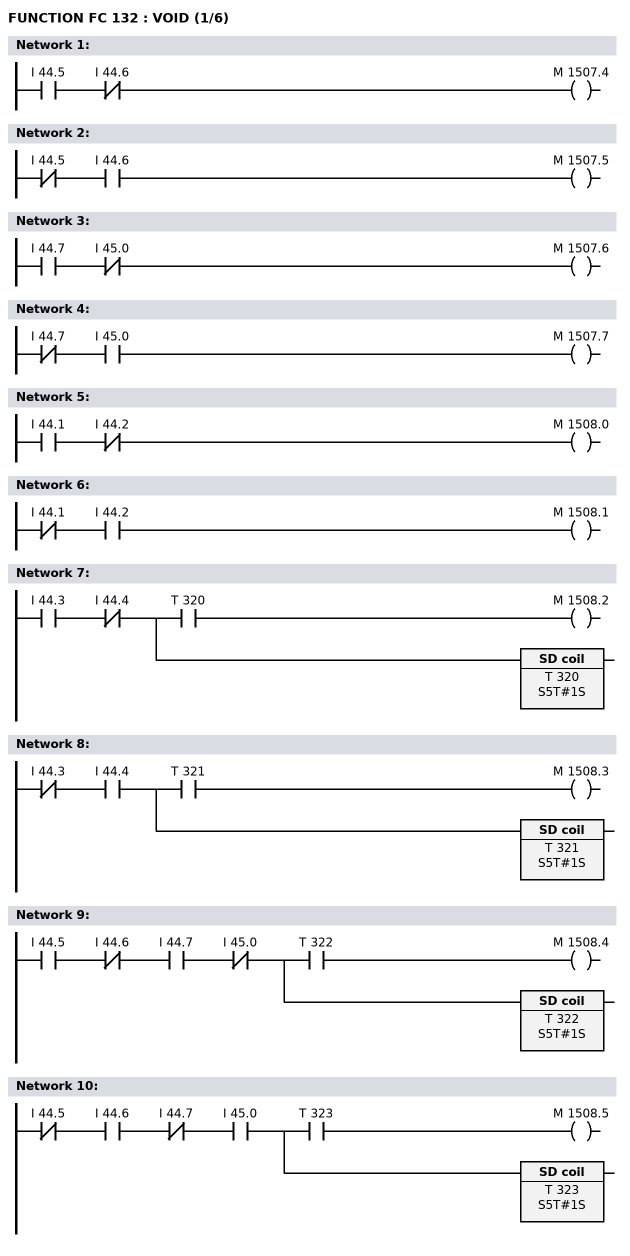

      A     I     44.5;
      AN    I     44.6;
      =     M   1507.4;
NETWORK
TITLE =

      AN    I     44.5;
      A     I     44.6;
      =     M   1507.5;
NETWORK
TITLE =

      A     I     44.7;
      AN    I     45.0;
      =     M   1507.6;
NETWORK
TITLE =

      AN    I     44.7;
      A     I     45.0;
      =     M   1507.7;
NETWORK
TITLE =

      A     I     44.1;
      AN    I     44.2;
      =     M   1508.0;
NETWORK
TITLE =

      AN    I     44.1;
      A     I     44.2;
      =     M   1508.1;
NETWORK
TITLE =

      A     I     44.3;
      AN    I     44.4;
      =     L      0.0;
      A     L      0.0;
      A     T    320;
      =     M   1508.2;
      A     L      0.0;
      BLD   102;
      L     S5T#1S;
      SD    T    320;
NETWORK
TITLE =

      AN    I     44.3;
      A     I     44.4;
      =     L      0.0;
      A     L      0.0;
      A     T    321;
      =     M   1508.3;
      A     L      0.0;
      BLD   102;
      L     S5T#1S;
      SD    T    321;
NETWORK
TITLE =

      A     I     44.5;
      AN    I     44.6;
      A     I     44.7;
      AN    I     45.0;
      =     L      0.0;
      A     L      0.0;
      A     T    322;
      =     M   1508.4;
      A     L      0.0;
      BLD   102;
      L     S5T#1S;
      SD    T    322;
NETWORK
TITLE =

      AN    I     44.5;
      A     I     44.6;
      AN    I     44.7;
      A     I     45.0;
      =     L      0.0;
      A     L      0.0;
      A     T    323;
      =     M   1508.5;
      A     L      0.0;
      BLD   102;
      L     S5T#1S;
      SD    T    323;
NETWORK
TITLE =
